(* IEC 61131-3 sources: Std_PalletMover/Class/MQTTClient_Interface (part 4) *)

            Logging_InterfLog(usLevel     :=  MQTTCLIENTINTERFACE_LOGGING_LEVEL_ERR,
                              dMsgGroup   :=  MQCLIINF_LOG_ERROR_DATAMAP_UNSUBSCRIBE_FAIL_MQCLI_GRP,
                              dMsgNbr     :=  MQCLIINF_LOG_ERROR_DATAMAP_UNSUBSCRIBE_FAIL_MQCLI_MSG,
                              pMsg        :=  MQCLIINF_LOG_ERROR_DATAMAP_UNSUBSCRIBE_FAIL_MQCLI_TEXT,
                              pPara1      :=  #tmpPara1,
                              pPara2      :=  #tmpPara2,
                              pPara3      :=  #pEntry^.pData$DINT,
                              pPara4      :=  NIL);

            pEntry^.State := DMSS_Error;
            pEntry^.udLastAction := ops.tAbsolute;

          end_if;

        //----------------------------------------------------
        //Wait for Unsubscribe confirmation
        //----------------------------------------------------
        t_e_DataMap_SubscribeStates::DMSS_WaitForUnsubscribe:

          if ops.tAbsolute - pEntry^.udLastAction >= cDataMapSubTimeout then

            //Create Log: DataMap Failed to subscribe Entry, Timeout. Moving On.

            tmpPara1 := to_dint(pEntry^.iMid);
            tmpPara2 := pEntry^.pData$DINT;

            Logging_InterfLog(usLevel     :=  MQTTCLIENTINTERFACE_LOGGING_LEVEL_ERR,
                              dMsgGroup   :=  MQCLIINF_LOG_ERROR_DATAMAP_UNSUBSCRIBE_FAIL_TIMEOUT_GRP,
                              dMsgNbr     :=  MQCLIINF_LOG_ERROR_DATAMAP_UNSUBSCRIBE_FAIL_TIMEOUT_MSG,
                              pMsg        :=  MQCLIINF_LOG_ERROR_DATAMAP_UNSUBSCRIBE_FAIL_TIMEOUT_TEXT,
                              pPara1      :=  #tmpPara1,
                              pPara2      :=  #cDataMapSubTimeout$DINT,
                              pPara3      :=  #tmpPara2,
                              pPara4      :=  NIL);

            pEntry^.State := DMSS_Unsubscribed;

          end_if;

        //----------------------------------------------------
        //Cleanup & Finish
        //----------------------------------------------------
        t_e_DataMap_SubscribeStates::DMSS_Unsubscribed:

          //Reset Mid
          pEntry^.iMid  := -1;

          //If the element must be removed do so, else return it to the original state
          if pEntry^.bRemove then

            if DataMap_RemoveElement_ByIndex( udIndex     :=  udCount,
                                              ElementType :=  DM_Subscribe) = FALSE then

               //Create Log: Failed to remove unsubscribed PubSub Entry from PubSub list.

               tmpPara1 := to_dint(pEntry^.iMid);
               tmpPara2 := to_dint(udCount);

               Logging_InterfLog(usLevel     :=  MQTTCLIENTINTERFACE_LOGGING_LEVEL_ERR,
                                 dMsgGroup   :=  MQCLIINF_LOG_ERROR_DATAMAP_UNSUBSCRIBE_FAIL_RMVE_LIST_GRP,
                                 dMsgNbr     :=  MQCLIINF_LOG_ERROR_DATAMAP_UNSUBSCRIBE_FAIL_RMVE_LIST_MSG,
                                 pMsg        :=  MQCLIINF_LOG_ERROR_DATAMAP_UNSUBSCRIBE_FAIL_RMVE_LIST_TEXT,
                                 pPara1      :=  #tmpPara1,
                                 pPara2      :=  #tmpPara2,
                                 pPara3      :=  NIL,
                                 pPara4      :=  NIL);

               pEntry^.State := DMSS_Error;
               pEntry^.udLastAction := ops.tAbsolute;

            end_if;

          //Return State to allow a resubscription.
          else

            pEntry^.State := DMSS_Ready;

          end_if;

        //----------------------------------------------------
        //Error Occurred
        //----------------------------------------------------
        t_e_DataMap_SubscribeStates::DMSS_Error:

          //Reset Mid
          pEntry^.iMid  := -1;

          //If the reset time is set, wait for reset
          if (cDataMapResetTimeout <> 0) &
             (ops.tAbsolute - pEntry^.udLastAction >= cDataMapResetTimeout) then

            pEntry^.State := DMSS_Ready;

          end_if;

      end_case;

    end_for;

  end_if;

END_FUNCTION

FUNCTION MQTTClient_Interface::DataMap_RemoveElement
	VAR_INPUT
		pElement 	: ^CHAR;
		ElementType 	: t_e_DataMap_ElementTypes;
	END_VAR
	VAR_OUTPUT
		bOK 	: BOOL;
	END_VAR
  VAR
  	udElementIndex : UDINT;
    pPublishEntry : ^t_s_DataMap_ElementEntry_Publish;
    pSubscribeEntry : ^t_s_DataMap_ElementEntry_Subscribe;
  END_VAR

  bOK := FALSE;
  udElementIndex := 0;

  if pElement = NIL then
    return;
  end_if;

  //==========================================
  //Based on the type of element
  //==========================================

  case ElementType of

    //-------------------------------------
    //Publish List
    //-------------------------------------
  	t_e_DataMap_ElementTypes::DM_Publish:

      if Config.pDataMapConfig^.udPublishElements > 0 then

        pPublishEntry := Config.pDataMapConfig^.Elements.pPublishEntries;

        for udElementIndex := 0 to Config.pDataMapConfig^.udPublishElements - 1 do

          if SigCLib.StrCmp(ps1:=#pPublishEntry^.aElement[0], ps2:=pElement) = 0 then
            bOK := DataMap_RemoveElement_ByIndex(udIndex:=udElementIndex, ElementType:=ElementType);
            exit;
          end_if;

          pPublishEntry$UDINT += sizeof(t_s_DataMap_ElementEntry_Publish);
        end_for;

      else
        return;
      end_if;

    //-------------------------------------
    //Subscribe List
    //-------------------------------------
  	t_e_DataMap_ElementTypes::DM_Subscribe:

      if Config.pDataMapConfig^.udSubscribeElements > 0 then

        pSubscribeEntry := Config.pDataMapConfig^.Elements.pSubscribeEntries;

        for udElementIndex := 0 to Config.pDataMapConfig^.udSubscribeElements - 1 do

          if SigCLib.StrCmp(ps1:=#pSubscribeEntry^.aElement[0], ps2:=pElement) = 0 then

            if pSubscribeEntry^.State = DMSS_Subscribed then
              pSubscribeEntry^.State    := DMSS_Unsubscribe;
              pSubscribeEntry^.bRemove  := TRUE;
              bOK                       := TRUE;
            end_if;

            exit;
          end_if;

          pSubscribeEntry$UDINT += sizeof(t_s_DataMap_ElementEntry_Subscribe);

        end_for;

      else
        return;
      end_if;

  end_case;

END_FUNCTION

FUNCTION MQTTClient_Interface::DataMap_RemoveElement_ByIndex
	VAR_INPUT
		udIndex 	: UDINT;
		ElementType 	: t_e_DataMap_ElementTypes;
	END_VAR
	VAR_OUTPUT
		bOK 	: BOOL;
	END_VAR
  VAR
  	tmpPara : DINT;
  END_VAR

  //Assume not OK
  bOK := FALSE;

  if Config.pDataMapConfig = NIL then
    //Create Log: Tried removing an entry from the DataMap, DataMap not inited.

    tmpPara := to_dint(udIndex);

    Logging_InterfLog(usLevel     :=  MQTTCLIENTINTERFACE_LOGGING_LEVEL_WARNING,
                      dMsgGroup   :=  MQCLIINF_LOG_WARNING_DATAMAP_REMOVE_FAILED_NOTINIT_GRP,
                      dMsgNbr     :=  MQCLIINF_LOG_WARNING_DATAMAP_REMOVE_FAILED_NOTINIT_MSG,
                      pMsg        :=  MQCLIINF_LOG_WARNING_DATAMAP_REMOVE_FAILED_NOTINIT_TEXT,
                      pPara1      :=  #tmpPara,
                      pPara2      :=  NIL,
                      pPara3      :=  NIL,
                      pPara4      :=  NIL);
    return;

  end_if;

  //========================================================
  //Based on the type of element - Find and remove the entry
  //========================================================
  case ElementType of

    //-------------------------------------
    //Publish List
    //-------------------------------------
  	t_e_DataMap_ElementTypes::DM_Publish:

      //If the index is ok
      if udIndex >= 0                                         &
         udIndex <  Config.pDataMapConfig^.udPublishElements  then

        //If this is the last entry, we don't need to copy any data
        if udIndex = Config.pDataMapConfig^.udPublishElements - 1 then

          Config.pDataMapConfig^.udPublishElements -= 1;

        //If this is not the last entry, the data has to be moved back
        else

          SigCLib.MemCpy( dst0  :=  (Config.pDataMapConfig^.Elements.pPublishEntries$UDINT + sizeof(t_s_DataMap_ElementEntry_Publish)*udIndex)$^void,
                          src0  :=  (Config.pDataMapConfig^.Elements.pPublishEntries$UDINT + sizeof(t_s_DataMap_ElementEntry_Publish)*(udIndex+1))$^void,
                          len0  :=  ((Config.pDataMapConfig^.udPublishElements-1) - udIndex)*sizeof(t_s_DataMap_ElementEntry_Publish));

          Config.pDataMapConfig^.udPublishElements -= 1;

        end_if;

        bOK := TRUE;
        return;

      else

        //Create Log: Tried removing an Entry from the DataMap with invalid Index.

        tmpPara := to_dint(udIndex);

        Logging_InterfLog(usLevel     :=  MQTTCLIENTINTERFACE_LOGGING_LEVEL_ERR,
                          dMsgGroup   :=  MQCLIINF_LOG_ERROR_DATAMAP_REMOVE_FAILED_INDEX_INV_GRP,
                          dMsgNbr     :=  MQCLIINF_LOG_ERROR_DATAMAP_REMOVE_FAILED_INDEX_INV_MSG,
                          pMsg        :=  MQCLIINF_LOG_ERROR_DATAMAP_REMOVE_FAILED_INDEX_INV_TEXT,
                          pPara1      :=  #tmpPara,
                          pPara2      :=  NIL,
                          pPara3      :=  NIL,
                          pPara4      :=  NIL);

      end_if;

    //-------------------------------------
    //Subscribe List
    //-------------------------------------
  	t_e_DataMap_ElementTypes::DM_Subscribe:

      //If the index is ok
      if udIndex >= 0 &
         udIndex <  Config.pDataMapConfig^.udSubscribeElements then

        if udIndex = Config.pDataMapConfig^.udSubscribeElements - 1 then
          Config.pDataMapConfig^.udSubscribeElements -= 1;
        else

          SigCLib.MemCpy( dst0  :=  (Config.pDataMapConfig^.Elements.pSubscribeEntries$UDINT + sizeof(t_s_DataMap_ElementEntry_Subscribe)*udIndex)$^void,
                          src0  :=  (Config.pDataMapConfig^.Elements.pSubscribeEntries$UDINT + sizeof(t_s_DataMap_ElementEntry_Subscribe)*(udIndex+1))$^void,
                          len0  :=  ((Config.pDataMapConfig^.udSubscribeElements-1) - udIndex)*sizeof(t_s_DataMap_ElementEntry_Subscribe));

          Config.pDataMapConfig^.udSubscribeElements -= 1;

        end_if;

        bOK := TRUE;
        return;

      else

        //Create Log: Tried removing an Entry from the DataMap with invalid Index.

        tmpPara := to_dint(udIndex);

        Logging_InterfLog(usLevel     :=  MQTTCLIENTINTERFACE_LOGGING_LEVEL_ERR,
                          dMsgGroup   :=  MQCLIINF_LOG_ERROR_DATAMAP_REMOVE_FAILED_INDEX_INV_GRP,
                          dMsgNbr     :=  MQCLIINF_LOG_ERROR_DATAMAP_REMOVE_FAILED_INDEX_INV_MSG,
                          pMsg        :=  MQCLIINF_LOG_ERROR_DATAMAP_REMOVE_FAILED_INDEX_INV_TEXT,
                          pPara1      :=  #tmpPara,
                          pPara2      :=  NIL,
                          pPara3      :=  NIL,
                          pPara4      :=  NIL);

      end_if;

  end_case;

END_FUNCTION

FUNCTION MQTTClient_Interface::DataMap_ResetStates
	VAR_OUTPUT
		bOK 	: BOOL;
	END_VAR
  VAR
  	udCount : UDINT;
    pSubElement : ^t_s_DataMap_ElementEntry_Subscribe;
    pPubElement : ^t_s_DataMap_ElementEntry_Publish;
  END_VAR

  //Assume Fail
  bOK := FALSE;

  //Reset Registered DataMap States
  if Config.pDataMapConfig then

    if Config.pDataMapConfig^.udSubscribeElements > 0 then
      pSubElement := Config.pDataMapConfig^.Elements.pSubscribeEntries;
      for udCount := 0 to Config.pDataMapConfig^.udSubscribeElements - 1 do
        pSubElement^.State := 0;
        pSubElement$UDINT += sizeof(t_s_DataMap_ElementEntry_Subscribe);
      end_for;
    end_if;

    if Config.pDataMapConfig^.udPublishElements > 0 then
      pPubElement:= Config.pDataMapConfig^.Elements.pPublishEntries;
      for udCount := 0 to Config.pDataMapConfig^.udPublishElements - 1 do
        pPubElement^.State := 0;
        pPubElement$UDINT += sizeof(t_s_DataMap_ElementEntry_Publish);
      end_for;
    end_if;

    bOK := TRUE;

  end_if;

END_FUNCTION

FUNCTION MQTTClient_Interface::DataMap_Return_Callback
	VAR_INPUT
		pThis 	: ^void;
		MsgType 	: MQTTClient_Interface::t_e_PubSubRetCodes;
		iMid 	: INT;
		iGrantedQoS 	: INT;
		pMessage 	: ^MQTTClient::t_s_MQTTMessage;
	END_VAR

  //Call Internal Method
  pThis$^MQTTClient_Interface^.DataMap_Return(MsgType     :=  MsgType,
                                              iMid        :=  iMid,
                                              iGrantedQoS :=  iGrantedQoS,
                                              pMessage    :=  pMessage);

END_FUNCTION

FUNCTION MQTTClient_Interface::DataMap_Clear

  if Config.pDataMapConfig                             &
     Config.pDataMapConfig^.Elements.pPublishEntries   &
     Config.pDataMapConfig^.Elements.pSubscribeEntries then

    Config.pDataMapConfig^.udPublishElements := 0;
    Config.pDataMapConfig^.udSubscribeElements := 0;

    sigclib_memset( dst :=  Config.pDataMapConfig^.Elements.pPublishEntries,
                    c   :=  0x00,
                    len :=  sizeof(t_s_DataMap_ElementEntry_Publish)*Config.pDataMapConfig^.udEntries);

    sigclib_memset( dst :=  Config.pDataMapConfig^.Elements.pSubscribeEntries,
                    c   :=  0x00,
                    len :=  sizeof(t_s_DataMap_ElementEntry_Subscribe)*Config.pDataMapConfig^.udEntries);

  end_if;

END_FUNCTION

FUNCTION MQTTClient_Interface::DataMap_Return
	VAR_INPUT
		MsgType 	: MQTTClient_Interface::t_e_PubSubRetCodes;
		iMid 	: INT;
		iGrantedQoS 	: INT;
		pMessage 	: ^MQTTClient::t_s_MQTTMessage;
	END_VAR
  VAR
  	udCount         : UDINT;
  	pArray          : ^void;
    pArrEntry       : ^void;
    udNumSubEntries : UDINT;
    pSubEntry       : ^t_s_DataMap_ElementEntry_Subscribe;
    pPubEntry       : ^t_s_DataMap_ElementEntry_Publish;
    bFound          : BOOL;
    udCopyLen       : UDINT;
    tmpPara1        : DINT;
    tmpPara2        : DINT;
    tmpPara3        : DINT;
    tmpPara4        : DINT;
    tmpData         : DINT; //Variable to contain the received 4 byte values temporarily, this avoids writing rubbish on the server
  END_VAR

  //Clear pSubEntries Pointer, Memory is malloc'd and set to this pointer if MsgType = PSRC_PublishReceived,
  //All exit paths must be observed to avoid a memory leak here.
  pArray := NIL;

  if Config.pDataMapConfig = NIL then
    //Create Log: Received Datamap Callback for DataMap Whilst DataMap is not Inited.

    tmpPara1 := to_dint(iMid);

    if pMessage <> NIL then
      tmpPara2 := to_dint(pMessage^.mid);
    else
      tmpPara2 := 16#FFFF;
    end_if;

    Logging_InterfLog(usLevel     :=  MQTTCLIENTINTERFACE_LOGGING_LEVEL_WARNING,
                      dMsgGroup   :=  MQCLIINF_LOG_WARNING_DATAMAP_CALLBACK_MAP_NOTINIT_GRP,
                      dMsgNbr     :=  MQCLIINF_LOG_WARNING_DATAMAP_CALLBACK_MAP_NOTINIT_MSG,
                      pMsg        :=  MQCLIINF_LOG_WARNING_DATAMAP_CALLBACK_MAP_NOTINIT_TEXT,
                      pPara1      :=  #tmpPara1,
                      pPara2      :=  #tmpPara2,
                      pPara3      :=  NIL,
                      pPara4      :=  NIL);

    return;
  end_if;

  bFound := FALSE;

  //======================================
  //Find the DataMap Entry with this Mid
  //======================================
  case MsgType of

    //------------------------------------------------
    //Disconnected
    //------------------------------------------------
  	PSRC_Disconnected:

      //Reset all the DataMap Entries

      return;

    //---------------------------------------------------------------------------
    //Subscribe Related, can only be: one entry (Mid Tracked) or all (Mid = -1)
    //---------------------------------------------------------------------------
  	PSRC_Subscribed, PSRC_Unsubscribed:

      pSubEntry := Config.pDataMapConfig^.Elements.pSubscribeEntries;
      if Config.pDataMapConfig^.udSubscribeElements > 0 then

        //If this is an unsubscribe all (iMid=-1), then simply unsubscribe all and return,
        //else find the entry to unsubscribe
        if iMid = -1 then

          for udCount := 0 to Config.pDataMapConfig^.udSubscribeElements - 1 do
            pSubEntry^.State := DMSS_Unsubscribed;
            pSubEntry$UDINT += sizeof(t_s_DataMap_ElementEntry_Subscribe);
          end_for;
          return;

        //This is a specific entry, step over all entries to find the matching entry.
        else

          for udCount := 0 to Config.pDataMapConfig^.udSubscribeElements - 1 do
            if pSubEntry^.iMid = iMid then
              bFound := TRUE;
              exit;
            end_if;
            pSubEntry$UDINT += sizeof(t_s_DataMap_ElementEntry_Subscribe);
          end_for;

        end_if;
      end_if;

    //----------------------------------------------------
    //Publish Related, Mid tracked, can only be one entry
    //----------------------------------------------------
  	PSRC_Published:

      pPubEntry := Config.pDataMapConfig^.Elements.pPublishEntries;
      for udCount := 0 to Config.pDataMapConfig^.udEntries - 1 do
        if pPubEntry^.iMid = iMid then
          pPubEntry^.iMid := -1;
          bFound := TRUE;
          exit;
        end_if;
        pPubEntry$UDINT += sizeof(t_s_DataMap_ElementEntry_Publish);
      end_for;

    //-------------------------------------------------------------------
    //Subscribe Related, Use Topic for relation, can be multiple entries
    //-------------------------------------------------------------------
    PSRC_PublishReceived:

      pArray := MQTTClient.MallocV1(size0 :=  sizeof(^void) * Config.pPubSubConfig^.PubSubList.udMaxEntries,
                                    mark0 :=  MQTTCLIENTINTERFACE_DEFAULT_MALLOC_MARK);

      //If the Malloc succeeded
      if pArray <> NIL then

        SigCLib.MemSet( dst :=  pArray,
                        c   :=  0x00,
                        len :=  sizeof(^void) * Config.pPubSubConfig^.PubSubList.udMaxEntries);

        udNumSubEntries := 0;
        pSubEntry := Config.pDataMapConfig^.Elements.pSubscribeEntries;
        pArrEntry := pArray;

        for udCount := 0 to Config.pDataMapConfig^.udSubscribeElements - 1 do

          //If this is not a stale entry and the topic matches, add to the list.
          if PubSub_TopicCompare(pStr:=pMessage^.topic, pWCString:=#pSubEntry^.aTopic[0]) then

            bFound := TRUE;
            pArrEntry^$UDINT := pSubEntry$UDINT;
            pArrEntry$UDINT += sizeof(^void);
            udNumSubEntries += 1;

          end_if;

          pSubEntry$UDINT += sizeof(t_s_DataMap_ElementEntry_Subscribe);

        end_for;

      //Malloc failed, we won't be able to deliver the message to the Application, report error.
      else

        tmpPara1 := to_dint(iMid);

        if pMessage <> NIL then
          tmpPara2 := to_dint(pMessage^.mid);
        else
          tmpPara2 := 16#FFFF;
        end_if;

        Logging_InterfLog(usLevel     :=  MQTTCLIENTINTERFACE_LOGGING_LEVEL_ERR,
                          dMsgGroup   :=  MQCLIINF_LOG_ERROR_DATAMAP_RETURN_NOMEM_ARRAY_GRP,
                          dMsgNbr     :=  MQCLIINF_LOG_ERROR_DATAMAP_RETURN_NOMEM_ARRAY_MSG,
                          pMsg        :=  MQCLIINF_LOG_ERROR_DATAMAP_RETURN_NOMEM_ARRAY_TEXT,
                          pPara1      :=  #tmpPara1,
                          pPara2      :=  #tmpPara2,
                          pPara3      :=  NIL,
                          pPara4      :=  NIL);

        return;

      end_if;

  end_case;

  if bFound = FALSE then
    //Create Log: Received DataMap Callback but did not find corresponding entry.

    tmpPara1 := to_dint(iMid);

    if pMessage <> NIL then
      tmpPara2 := to_dint(pMessage^.mid);
    else
      tmpPara2 := 16#FFFF;
    end_if;

    Logging_InterfLog(usLevel     :=  MQTTCLIENTINTERFACE_LOGGING_LEVEL_ERR,
                      dMsgGroup   :=  MQCLIINF_LOG_WARNING_DATAMAP_CALLBACK_ENTRY_NOTFOUND_GRP,
                      dMsgNbr     :=  MQCLIINF_LOG_WARNING_DATAMAP_CALLBACK_ENTRY_NOTFOUND_MSG,
                      pMsg        :=  MQCLIINF_LOG_WARNING_DATAMAP_CALLBACK_ENTRY_NOTFOUND_TEXT,
                      pPara1      :=  #tmpPara1,
                      pPara2      :=  #tmpPara2,
                      pPara3      :=  NIL,
                      pPara4      :=  NIL);

    //If the pSubEntries Pointer is set, free
    if pArray then
      MQTTClient.Free(mptr:=pArray);
      pArray := NIL;
    end_if;

    return;
  end_if;

  //=====================================================
  //Based on the type of message, edit the DataMap
  //=====================================================
  case MsgType of

    //------------------------------------------------
    //Subscribe completed, check and advance
    //------------------------------------------------
    t_e_PubSubRetCodes::PSRC_Subscribed:

      //if the QoS is invalid, set state and log
      if iGrantedQoS < MQTT_PROT_QOS_MIN |
         iGrantedQoS > MQTT_PROT_QOS_MAX then
        //Create Log: DataMap Element Failed to Subscribe, Returned QoS Invalid, Element=XXXX Granted=XX, Requested=XX

        tmpPara1 := to_dint(iMid);

        if pMessage <> NIL then
          tmpPara2 := to_dint(pMessage^.mid);
        else
          tmpPara2 := 16#FFFF;
        end_if;

        tmpPara3 := to_dint(iGrantedQoS);

        if pSubEntry <> NIL then
          tmpPara4 := to_dint(pSubEntry^.iQoS);
        else
          tmpPara4 := 16#FFFF;
        end_if;

        Logging_InterfLog(usLevel     :=  MQTTCLIENTINTERFACE_LOGGING_LEVEL_ERR,
                          dMsgGroup   :=  MQCLIINF_LOG_ERROR_DATAMAP_SUB_CONF_WRONG_QOS_GRP,
                          dMsgNbr     :=  MQCLIINF_LOG_ERROR_DATAMAP_SUB_CONF_WRONG_QOS_MSG,
                          pMsg        :=  MQCLIINF_LOG_ERROR_DATAMAP_SUB_CONF_WRONG_QOS_TEXT,
                          pPara1      :=  #tmpPara1,
                          pPara2      :=  #tmpPara2,
                          pPara3      :=  #tmpPara3,
                          pPara4      :=  #tmpPara4);

        pSubEntry^.State := DMSS_Error;
        return;
      end_if;

      //If the Entry is not in the correct state
      if pSubEntry^.State <> DMSS_WaitForSubscribe then
        //Create Log: DataMap Element failed to Subscribe, Subscription returned valid but the Element State was invalid, Element=XXXX, Granted QoS=XX

        tmpPara1 := to_dint(iMid);

        if pMessage <> NIL then
          tmpPara2 := to_dint(pMessage^.mid);
        else
          tmpPara2 := 16#FFFF;
        end_if;

        tmpPara3 := to_dint(pSubEntry^.State);

        Logging_InterfLog(usLevel     :=  MQTTCLIENTINTERFACE_LOGGING_LEVEL_ERR,
                          dMsgGroup   :=  MQCLIINF_LOG_WARNING_DATAMAP_SUB_CONFD_WRONG_STATE_GRP,
                          dMsgNbr     :=  MQCLIINF_LOG_WARNING_DATAMAP_SUB_CONFD_WRONG_STATE_MSG,
                          pMsg        :=  MQCLIINF_LOG_WARNING_DATAMAP_SUB_CONFD_WRONG_STATE_TEXT,
                          pPara1      :=  #tmpPara1,
                          pPara2      :=  #tmpPara2,
                          pPara3      :=  #tmpPara3,
                          pPara4      :=  NIL);

        pSubEntry^.State := DMSS_Error;
        return;

      end_if;

      //If QoS does not match then log the difference and update
      if iGrantedQoS <> pSubEntry^.iQoS then
        //Create Log: DataMap Element Granted QoS differs from Requested, Element=XXXX Granted=XX, Requested=XX

        tmpPara1 := to_dint(iMid);

        if pMessage <> NIL then
          tmpPara2 := to_dint(pMessage^.mid);
        else
          tmpPara2 := 16#FFFF;
        end_if;

        tmpPara3 := to_dint(iGrantedQoS);

        if pSubEntry <> NIL then
          tmpPara4 := to_dint(pSubEntry^.iQoS);
        else
          tmpPara4 := 16#FFFF;
        end_if;

        Logging_InterfLog(usLevel     :=  MQTTCLIENTINTERFACE_LOGGING_LEVEL_INFO,
                          dMsgGroup   :=  MQCLIINF_LOG_INFO_DATAMAP_SUB_CONFD_QOS_DIFFERS_GRP,
                          dMsgNbr     :=  MQCLIINF_LOG_INFO_DATAMAP_SUB_CONFD_QOS_DIFFERS_MSG,
                          pMsg        :=  MQCLIINF_LOG_INFO_DATAMAP_SUB_CONFD_QOS_DIFFERS_TEXT,
                          pPara1      :=  #tmpPara1,
                          pPara2      :=  #tmpPara2,
                          pPara3      :=  #tmpPara3,
                          pPara4      :=  #tmpPara4);

        pSubEntry^.iQoS := iGrantedQoS;
      end_if;

      pSubEntry^.State := DMSS_Subscribed;

    //------------------------------------------------
    //Unsubscribe completed, check and advance
    //------------------------------------------------
    t_e_PubSubRetCodes::PSRC_Unsubscribed:

      //Create Log: DataMap Element Unsubscribed, Element=XXXX

      tmpPara1 := to_dint(iMid);

      if pMessage <> NIL then
        tmpPara2 := to_dint(pMessage^.mid);
      else
        tmpPara2 := 16#FFFF;
      end_if;

      Logging_InterfLog(usLevel     :=  MQTTCLIENTINTERFACE_LOGGING_LEVEL_INFO,
                        dMsgGroup   :=  MQCLIINF_LOG_INFO_DATAMAP_UNSUB_CONFD_GRP,
                        dMsgNbr     :=  MQCLIINF_LOG_INFO_DATAMAP_UNSUB_CONFD_MSG,
                        pMsg        :=  MQCLIINF_LOG_INFO_DATAMAP_UNSUB_CONFD_TEXT,
                        pPara1      :=  #tmpPara1,
                        pPara2      :=  #tmpPara2,
                        pPara3      :=  NIL,
                        pPara4      :=  NIL);

      pSubEntry^.State := DMSS_Unsubscribed;

    //------------------------------------------------
    //Publish Received, Set Data
    //------------------------------------------------
    t_e_PubSubRetCodes::PSRC_PublishReceived:

      if pMessage then

        //Step over all the entries found and process the message
        if udNumSubEntries > 0 then

          for udCount := 0 to udNumSubEntries - 1 do

            //pSubEntry := aSubEntries[udCount];
            pSubEntry$UDINT := (pArray$UDINT + sizeof(^void)*udCount);
            pSubEntry := pSubEntry^$^t_s_DataMap_ElementEntry_Subscribe;

            //======================================
            //Set the data based on the type
            //======================================
            case pSubEntry^.DataType of
              //----------------------
              //4 Bytes
              //----------------------
              t_e_DataMap_DataTypes::DD_UDINT:

                udCopyLen := pMessage^.payloadlen;

                if udCopyLen > sizeof(UDINT) then
                  //Create Log: More data received than is able to be fit into Datamap element, data truncated

                  tmpPara1 := to_dint(iMid);

                  if pMessage <> NIL then
                    tmpPara2 := to_dint(pMessage^.mid);
                  else
                    tmpPara2 := 16#FFFF;
                  end_if;

                  Logging_InterfLog(usLevel     :=  MQTTCLIENTINTERFACE_LOGGING_LEVEL_WARNING,
                                    dMsgGroup   :=  MQCLIINF_LOG_WARNING_DATAMAP_DATA_TRUNCATED_UDINT_GRP,
                                    dMsgNbr     :=  MQCLIINF_LOG_WARNING_DATAMAP_DATA_TRUNCATED_UDINT_MSG,
                                    pMsg        :=  MQCLIINF_LOG_WARNING_DATAMAP_DATA_TRUNCATED_UDINT_TEXT,
                                    pPara1      :=  #tmpPara1,
                                    pPara2      :=  #tmpPara2,
                                    pPara3      :=  #udCopyLen$DINT,
                                    pPara4      :=  NIL);

                  udCopyLen := sizeof(UDINT);

                end_if;

                tmpData := 0;
                SigCLib.MemCpy( dst0  :=  #tmpData,
                                src0  :=  pMessage^.payload,
                                len0  :=  pMessage^.payloadlen);

                WR( pt    :=  pSubEntry^.pData,
                    dData :=  tmpData$DINT);

              //----------------------
              //4 Bytes
              //----------------------
              t_e_DataMap_DataTypes::DD_DINT:

                udCopyLen := pMessage^.payloadlen;

                if udCopyLen > sizeof(DINT) then
                  //Create Log: More data received than is able to be fit into Datamap element, data truncated

                  tmpPara1 := to_dint(iMid);

                  if pMessage <> NIL then
                    tmpPara2 := to_dint(pMessage^.mid);
                  else
                    tmpPara2 := 16#FFFF;
                  end_if;

                  Logging_InterfLog(usLevel     :=  MQTTCLIENTINTERFACE_LOGGING_LEVEL_WARNING,
                                    dMsgGroup   :=  MQCLIINF_LOG_WARNING_DATAMAP_DATA_TRUNCATED_DINT_GRP,
                                    dMsgNbr     :=  MQCLIINF_LOG_WARNING_DATAMAP_DATA_TRUNCATED_DINT_MSG,
                                    pMsg        :=  MQCLIINF_LOG_WARNING_DATAMAP_DATA_TRUNCATED_DINT_TEXT,
                                    pPara1      :=  #tmpPara1,
                                    pPara2      :=  #tmpPara2,
                                    pPara3      :=  #udCopyLen$DINT,
                                    pPara4      :=  NIL);

                  udCopyLen := sizeof(UDINT);

                end_if;

                tmpData := 0;
                SigCLib.MemCpy( dst0  :=  #tmpData,
                                src0  :=  pMessage^.payload,
                                len0  :=  pMessage^.payloadlen);

                WR( pt    :=  pSubEntry^.pData,
                    dData :=  tmpData$DINT);

              //----------------------
              //4 Bytes
              //----------------------
              t_e_DataMap_DataTypes::DD_REAL:

                udCopyLen := pMessage^.payloadlen;

                if udCopyLen > sizeof(REAL) then
                  //Create Log: More data received than is able to be fit into Datamap element, data truncated

                  tmpPara1 := to_dint(iMid);

                  if pMessage <> NIL then
                    tmpPara2 := to_dint(pMessage^.mid);
                  else
                    tmpPara2 := 16#FFFF;
                  end_if;

                  Logging_InterfLog(usLevel     :=  MQTTCLIENTINTERFACE_LOGGING_LEVEL_WARNING,
                                    dMsgGroup   :=  MQCLIINF_LOG_WARNING_DATAMAP_DATA_TRUNCATED_REAL_GRP,
                                    dMsgNbr     :=  MQCLIINF_LOG_WARNING_DATAMAP_DATA_TRUNCATED_REAL_MSG,
                                    pMsg        :=  MQCLIINF_LOG_WARNING_DATAMAP_DATA_TRUNCATED_REAL_TEXT,
                                    pPara1      :=  #tmpPara1,
                                    pPara2      :=  #tmpPara2,
                                    pPara3      :=  #udCopyLen$DINT,
                                    pPara4      :=  NIL);

                  udCopyLen := sizeof(UDINT);

                end_if;

                tmpData := 0;
                SigCLib.MemCpy( dst0  :=  #tmpData,
                                src0  :=  pMessage^.payload,
                                len0  :=  pMessage^.payloadlen);

                WR( pt    :=  pSubEntry^.pData,
                    dData :=  tmpData$DINT);

              //----------------------
              //Dynamic Size
              //----------------------
              t_e_DataMap_DataTypes::DD_String:

                pSubEntry^.pData$^StringInternal^.WriteDataOff(udLen :=  pMessage^.payloadlen,
                                                               udOff :=  0,
                                                               pData :=  pMessage^.payload$^USINT);

            end_case;

          end_for;

        end_if;

      else

        //Create Log: DataMap Received PublishReceived Callback from MQTTClientInterface but no message was set

        tmpPara1 := to_dint(iMid);

        if pMessage <> NIL then
          tmpPara2 := to_dint(pMessage^.mid);
        else
          tmpPara2 := 16#FFFF;
        end_if;

        Logging_InterfLog(usLevel     :=  MQTTCLIENTINTERFACE_LOGGING_LEVEL_WARNING,
                          dMsgGroup   :=  MQCLIINF_LOG_WARNING_DATAMAP_DATA_EMPTY_GRP,
                          dMsgNbr     :=  MQCLIINF_LOG_WARNING_DATAMAP_DATA_EMPTY_MSG,
                          pMsg        :=  MQCLIINF_LOG_WARNING_DATAMAP_DATA_EMPTY_TEXT,
                          pPara1      :=  #tmpPara1,
                          pPara2      :=  #tmpPara2,
                          pPara3      :=  NIL,
                          pPara4      :=  NIL);

      end_if;

      //If the pSubEntries Pointer is set, free
      if pArray then
        MQTTClient.Free(mptr:=pArray);
        pArray := NIL;
      end_if;

    //------------------------------------------------
    //Publish Complete
    //------------------------------------------------
    t_e_PubSubRetCodes::PSRC_Published:

      pPubEntry^.bPublishComplete := TRUE;

      return;

  end_case;

END_FUNCTION

//================================================================================================================================================================
//-------------------------------------------------------------------END OF DATAMAP METHODS-----------------------------------------------------------------------
//================================================================================================================================================================

//================================================================================================================================================================
//------------------------------------------------------------------------CALLBACK METHODS------------------------------------------------------------------------
//================================================================================================================================================================
FUNCTION MQTTClient_Interface::Callback_OnConnectWithFlags
	VAR_INPUT
		pThis 	: ^void;
		retCode 	: INT;
    flags   : BYTE;
	END_VAR

  if pThis then
    pThis$^MQTTClient_Interface^.OnConnectWithFlags(retCode:=retCode,flags:=flags);
  end_if;

END_FUNCTION

FUNCTION MQTTClient_Interface::Callback_OnDisconnect
	VAR_INPUT
		pThis 	: ^void;
		retCode 	: INT;
	END_VAR

  if pThis then
    pThis$^MQTTClient_Interface^.OnDisconnect(retCode:=retCode);
  end_if;

END_FUNCTION

FUNCTION MQTTClient_Interface::Callback_OnPublish
	VAR_INPUT
		pThis 	: ^void;
		mid 	: INT;
	END_VAR

  if pThis then
    pThis$^MQTTClient_Interface^.OnPublish(mid:=mid);
  end_if;

END_FUNCTION

FUNCTION MQTTClient_Interface::Callback_OnMessage
	VAR_INPUT
		pThis 	: ^void;
		pMessage 	: ^MQTTClient::t_s_MQTTMessage;
	END_VAR

  if pThis then
    pThis$^MQTTClient_Interface^.OnMessage(pMessage:=pMessage);
  end_if;

END_FUNCTION

FUNCTION MQTTClient_Interface::Callback_OnSubscribe
	VAR_INPUT
		pThis 	: ^void;
		mid 	: INT;
		qos_count 	: INT;
		granted_qos 	: ^INT;
	END_VAR

  if pThis then
    pThis$^MQTTClient_Interface^.OnSubscribe( mid         :=  mid,
                                              qos_count   := qos_count,
                                              granted_qos := granted_qos);
  end_if;

END_FUNCTION

FUNCTION MQTTClient_Interface::Callback_OnUnsubscribe
	VAR_INPUT
		pThis 	: ^void;
		mid 	: INT;
	END_VAR

  if pThis then
    pThis$^MQTTClient_Interface^.OnUnsubscribe(mid:=mid);
  end_if;

END_FUNCTION

FUNCTION MQTTClient_Interface::Callback_OnLog
	VAR_INPUT
		pThis 	: ^void;
		level 	: INT;
		pStr 	: ^CHAR;
	END_VAR

  if pThis then
    pThis$^MQTTClient_Interface^.OnLog( level :=  level,
                                        pStr  :=  pStr);
  end_if;

END_FUNCTION

FUNCTION MQTTClient_Interface::Callback_OnLog_WithDetail
	VAR_INPUT
		pThis 	    : ^void;
		usLevel 	  : USINT;
		dMsgGroup 	: DINT;
		dMsgNbr 	  : DINT;
		pMsg 	      : ^CHAR;
		pPara1 	    : ^DINT;
		pPara2 	    : ^DINT;
		pPara3 	    : ^DINT;
		pPara4 	    : ^DINT;
	END_VAR

  if pThis then

    pThis$^MQTTClient_Interface^.OnLog_WithDetail(usLevel   := usLevel,
                                                  dMsgGroup := dMsgGroup,
                                                  dMsgNbr   := dMsgNbr,
                                                  pMsg      := pMsg,
                                                  pPara1    := pPara1,
                                                  pPara2    := pPara2,
                                                  pPara3    := pPara3,
                                                  pPara4    := pPara4);

  end_if;

END_FUNCTION

FUNCTION MQTTClient_Interface::OnConnectWithFlags
	VAR_INPUT
		retCode 	: INT;
		flags 	  : BYTE;
	END_VAR
  VAR
  	tmpPara, tmpPara2 : DINT;
  END_VAR

  //=================================
  //Internal Actions

  //If in the correct state, process the Connect message, else log
  if InterfaceState = MCIS_WaitForConnection |
     InterfaceState = MCIS_Reconnecting      then

    if retCode = MQTT_PROT_CONNACK_RET_CONNACCEPTED then

      InterfaceState := MCIS_Connected;

      //Handle Flags

        //Tell the Subscribed entities that they have been unsubscribed.
        if  SessionPresent.Read() = 0 then
          MQTT_SetCleanSession();
        end_if;

      //Create Log: Connected

      tmpPara := to_dint(retCode);
      tmpPara2 := to_dint(flags);

      Logging_InterfLog(usLevel     :=  MQTTCLIENTINTERFACE_LOGGING_LEVEL_INFO,
                        dMsgGroup   :=  MQCLIINF_LOG_INFO_CONNECTION_CONNECTED_GRP,
                        dMsgNbr     :=  MQCLIINF_LOG_INFO_CONNECTION_CONNECTED_MSG,
                        pMsg        :=  MQCLIINF_LOG_INFO_CONNECTION_CONNECTED_TEXT,
                        pPara1      :=  #tmpPara,
                        pPara2      :=  #tmpPara2,
                        pPara3      :=  NIL,
                        pPara4      :=  NIL);

      Diagnostic_Event( Event   :=  DL_Connect,
                        udValue :=  0);

    elsif retCode = MQTT_PROT_CONNACK_RET_PROTVERSION then

      //Create Log: Connection Failed, Protocol Versions Mismatch

      tmpPara := to_dint(retCode);

      Logging_InterfLog(usLevel     :=  MQTTCLIENTINTERFACE_LOGGING_LEVEL_ERR,
                        dMsgGroup   :=  MQCLIINF_LOG_ERROR_CONNECTION_CONN_FAIL_VER_GRP,
                        dMsgNbr     :=  MQCLIINF_LOG_ERROR_CONNECTION_CONN_FAIL_VER_MSG,
                        pMsg        :=  MQCLIINF_LOG_ERROR_CONNECTION_CONN_FAIL_VER_TEXT,
                        pPara1      :=  #tmpPara,
                        pPara2      :=  NIL,
                        pPara3      :=  NIL,
                        pPara4      :=  NIL);

      InterfaceState := MCIS_Error;

    elsif retCode = MQTT_PROT_CONNACK_RET_ID_REJECTED then

      //Create Log: Connection Failed, ClientID Rejected

      tmpPara := to_dint(retCode);

      Logging_InterfLog(usLevel     :=  MQTTCLIENTINTERFACE_LOGGING_LEVEL_ERR,
                        dMsgGroup   :=  MQCLIINF_LOG_ERROR_CONNECTION_CONN_FAIL_CLIENTID_GRP,
                        dMsgNbr     :=  MQCLIINF_LOG_ERROR_CONNECTION_CONN_FAIL_CLIENTID_MSG,
                        pMsg        :=  MQCLIINF_LOG_ERROR_CONNECTION_CONN_FAIL_CLIENTID_TEXT,
                        pPara1      :=  #tmpPara,
                        pPara2      :=  NIL,
                        pPara3      :=  NIL,
                        pPara4      :=  NIL);

      InterfaceState := MCIS_Error;

    elsif retCode = MQTT_PROT_CONNACK_RET_SERVER_UNAVAIL then

      //Create Log: Connection Failed, Server unavailable

      tmpPara := to_dint(retCode);

      Logging_InterfLog(usLevel     :=  MQTTCLIENTINTERFACE_LOGGING_LEVEL_ERR,
                        dMsgGroup   :=  MQCLIINF_LOG_ERROR_CONNECTION_CONN_FAIL_SERV_UNAV_GRP,
                        dMsgNbr     :=  MQCLIINF_LOG_ERROR_CONNECTION_CONN_FAIL_SERV_UNAV_MSG,
                        pMsg        :=  MQCLIINF_LOG_ERROR_CONNECTION_CONN_FAIL_SERV_UNAV_TEXT,
                        pPara1      :=  #tmpPara,
                        pPara2      :=  NIL,
                        pPara3      :=  NIL,
                        pPara4      :=  NIL);

      InterfaceState := MCIS_Error;

    elsif retCode = MQTT_PROT_CONNACK_RET_USN_PASS then

      //Create Log: Connection Failed, Username and/or Password incorrect

      tmpPara := to_dint(retCode);

      Logging_InterfLog(usLevel     :=  MQTTCLIENTINTERFACE_LOGGING_LEVEL_ERR,
                        dMsgGroup   :=  MQCLIINF_LOG_ERROR_CONNECTION_CONN_FAIL_USNPWD_GRP,
                        dMsgNbr     :=  MQCLIINF_LOG_ERROR_CONNECTION_CONN_FAIL_USNPWD_MSG,
                        pMsg        :=  MQCLIINF_LOG_ERROR_CONNECTION_CONN_FAIL_USNPWD_TEXT,
                        pPara1      :=  #tmpPara,
                        pPara2      :=  NIL,
                        pPara3      :=  NIL,
                        pPara4      :=  NIL);

      InterfaceState := MCIS_Error;

    elsif retCode = MQTT_PROT_CONNACK_RET_NOT_AUTHD then

      //Create Log: Connection Failed, Not authorised

      tmpPara := to_dint(retCode);

      Logging_InterfLog(usLevel     :=  MQTTCLIENTINTERFACE_LOGGING_LEVEL_ERR,
                        dMsgGroup   :=  MQCLIINF_LOG_ERROR_CONNECTION_CONN_FAIL_NOT_AUTH_GRP,
                        dMsgNbr     :=  MQCLIINF_LOG_ERROR_CONNECTION_CONN_FAIL_NOT_AUTH_MSG,
                        pMsg        :=  MQCLIINF_LOG_ERROR_CONNECTION_CONN_FAIL_NOT_AUTH_TEXT,
                        pPara1      :=  #tmpPara,
                        pPara2      :=  NIL,
                        pPara3      :=  NIL,
                        pPara4      :=  NIL);

      InterfaceState := MCIS_Error;

    end_if;

  //Not expecting callback
  else

    //Create Log: Unexpected Connect Callback Received

    tmpPara := to_dint(retCode);

    Logging_InterfLog(usLevel     :=  MQTTCLIENTINTERFACE_LOGGING_LEVEL_ERR,
                      dMsgGroup   :=  MQCLIINF_LOG_WARNING_CONNECTION_CONN_CALLBACK_UNEXP_GRP,
                      dMsgNbr     :=  MQCLIINF_LOG_WARNING_CONNECTION_CONN_CALLBACK_UNEXP_MSG,
                      pMsg        :=  MQCLIINF_LOG_WARNING_CONNECTION_CONN_CALLBACK_UNEXP_TEXT,
                      pPara1      :=  #tmpPara,
                      pPara2      :=  NIL,
                      pPara3      :=  NIL,
                      pPara4      :=  NIL);

  end_if;

  //=================================
  //Signed in Objects

END_FUNCTION

FUNCTION MQTTClient_Interface::OnDisconnect
	VAR_INPUT
		retCode 	: INT;
	END_VAR
  VAR
  	udCount : UDINT;
    tmpPara : DINT;
    pEntry  : ^t_s_PubSubEntry;
  END_VAR

  //=================================
  //Internal Actions

  //=============================================
  //Handle Disconnect Message according to state
  //=============================================
  case InterfaceState of

    //------------------------------------------------------------------
    //Was Connected and then Disconnected, advance State
    //------------------------------------------------------------------
  	MQTTClient_Interface::t_e_MQTTClientStates::MCIS_Connected:

      //User Request, Go to ready
      if retCode = MQTTCLIENT_DISCONNECT_RETCODE_USER then

        InterfaceState := MCIS_Ready;
        //Create Log: MQTT Interface Successfully Disconnected due to user request

        tmpPara := to_dint(retcode);

        Logging_InterfLog(usLevel     :=  MQTTCLIENTINTERFACE_LOGGING_LEVEL_INFO,
                          dMsgGroup   :=  MQCLIINF_LOG_INFO_CONNECTION_DISCONNECTED_GRP,
                          dMsgNbr     :=  MQCLIINF_LOG_INFO_CONNECTION_DISCONNECTED_MSG,
                          pMsg        :=  MQCLIINF_LOG_INFO_CONNECTION_DISCONNECTED_TEXT,
                          pPara1      :=  #tmpPara,
                          pPara2      :=  NIL,
                          pPara3      :=  NIL,
                          pPara4      :=  NIL);

      //Unexpected, wait for connection
      elsif retCode = MQTTCLIENT_DISCONNECT_RETCODE_UNEXP then

        InterfaceState := MCIS_Reconnecting;
        //Diagnostic Info:
        Diagnostic_Event( Event   :=  DL_ConnectRetry,
                          udValue :=  0);

        //Create Log: MQTT Interface Disconnected Unexpectedly, Waiting for reconnection.

        tmpPara := to_dint(retcode);

        Logging_InterfLog(usLevel     :=  MQTTCLIENTINTERFACE_LOGGING_LEVEL_WARNING,
                          dMsgGroup   :=  MQCLIINF_LOG_ERROR_CONNECTION_DISCONN_UNEXP_GRP,
                          dMsgNbr     :=  MQCLIINF_LOG_ERROR_CONNECTION_DISCONN_UNEXP_MSG,
                          pMsg        :=  MQCLIINF_LOG_ERROR_CONNECTION_DISCONN_UNEXP_TEXT,
                          pPara1      :=  #tmpPara,
                          pPara2      :=  NIL,
                          pPara3      :=  NIL,
                          pPara4      :=  NIL);

      //Undefined RetCode, Log, Error
      else

        //Create Log: MQTT Client Diconnected with undefined disconnect code.

        tmpPara := to_dint(retcode);

        Logging_InterfLog(usLevel     :=  MQTTCLIENTINTERFACE_LOGGING_LEVEL_ERR,
                          dMsgGroup   :=  MQCLIINF_LOG_ERROR_CONNECTION_DISCONN_UNKNOWN_CODE_GRP,
                          dMsgNbr     :=  MQCLIINF_LOG_ERROR_CONNECTION_DISCONN_UNKNOWN_CODE_MSG,
                          pMsg        :=  MQCLIINF_LOG_ERROR_CONNECTION_DISCONN_UNKNOWN_CODE_TEXT,
                          pPara1      :=  #tmpPara,
                          pPara2      :=  NIL,
                          pPara3      :=  NIL,
                          pPara4      :=  NIL);

        InterfaceState := MCIS_Error;

      end_if;

    //------------------------------------------------------------------
    //Unexpected callback
    //------------------------------------------------------------------
    else

      //Create Log: Unexpected Disconnect Message Received from MQTT Client

      tmpPara := to_dint(retcode);

      Logging_InterfLog(usLevel     :=  MQTTCLIENTINTERFACE_LOGGING_LEVEL_WARNING,
                        dMsgGroup   :=  MQCLIINF_LOG_WARNING_CONNECTION_DISCONN_CALLBACK_UNEXP_GRP,
                        dMsgNbr     :=  MQCLIINF_LOG_WARNING_CONNECTION_DISCONN_CALLBACK_UNEXP_MSG,
                        pMsg        :=  MQCLIINF_LOG_WARNING_CONNECTION_DISCONN_CALLBACK_UNEXP_TEXT,
                        pPara1      :=  #tmpPara,
                        pPara2      :=  NIL,
                        pPara3      :=  NIL,
                        pPara4      :=  NIL);

      InterfaceState := MCIS_Error;

  end_case;

  //Perform the disconnect callbacks for the items in the pubsub list
  if Config.pPubSubConfig &
     Config.pPubSubConfig^.PubSubList.udNumEntries > 0 then

    for udCount := 0 to Config.pPubSubConfig^.PubSubList.udNumEntries -1 do

      pEntry := (Config.pPubSubConfig^.PubSubList.pEntries$UDINT + sizeof(t_s_PubSubEntry)*udCount)$^t_s_PubSubEntry;

      if pEntry^.Callback.pThis    &
         pEntry^.Callback.pMethod  then

        pEntry^.Callback.pMethod$PubSub_Callback( pThis       :=  pEntry^.Callback.pThis,
                                                  MsgType     :=  PSRC_Disconnected,
                                                  iMid        :=  -1,
                                                  iGrantedQoS :=  -1,
                                                  pMessage    :=  NIL);

       //If this is the MQTTTopic Class
      elsif pEntry^.Callback.pThis          &
            pEntry^.Callback.pMethod = NIL  then

        pEntry^.Callback.pThis$^MQTTTopic^.PubSubData(MsgType     :=  PSRC_Disconnected,
                                                      iMid        :=  -1,
                                                      iGrantedQoS :=  -1,
                                                      pMessage    :=  NIL);

      end_if;

    end_for;

  end_if;

END_FUNCTION

FUNCTION MQTTClient_Interface::OnPublish
	VAR_INPUT
		mid 	: INT;
	END_VAR
  VAR
  	udCount : UDINT;
    pEntry : ^t_s_PubSubEntry;
    tmpPara : DINT;
  END_VAR

  //If there aren't any Subscribe elements in the Subscribe List | Mem not OK
  if Config.pPubSubConfig^.PubSubList.udNumEntries = 0 then
    //Create Log: Received Publish confirm from MQTTClient without having any elements in the subscription list, ignored.

    tmpPara := to_dint(mid);

    Logging_InterfLog(usLevel     :=  MQTTCLIENTINTERFACE_LOGGING_LEVEL_ERR,
                      dMsgGroup   :=  MQCLIINF_LOG_ERROR_PUBLISH_UNEXPECTED_PUB_CONF_NOTINIT_GRP,
                      dMsgNbr     :=  MQCLIINF_LOG_ERROR_PUBLISH_UNEXPECTED_PUB_CONF_NOTINIT_MSG,
                      pMsg        :=  MQCLIINF_LOG_ERROR_PUBLISH_UNEXPECTED_PUB_CONF_NOTINIT_TEXT,
                      pPara1      :=  #tmpPara,
                      pPara2      :=  NIL,
                      pPara3      :=  NIL,
                      pPara4      :=  NIL);
    return;
  end_if;

  //Step over the entries to find the responsible one
  pEntry := Config.pPubSubConfig^.PubSubList.pEntries;

  for udCount := 0 to Config.pPubSubConfig^.PubSubList.udNumEntries - 1 do

    if pEntry^.iMid = mid &
       pEntry^.EntryType = PSE_Publish then

//      if pEntry^.EntryType <> PSE_Publish then
//        //Create Log: Received a Publish confirmation for a non publish item in the pubsub list, ignored.
//
//        tmpPara := to_dint(mid);
//
//        Logging_InterfLog(usLevel     :=  MQTTCLIENTINTERFACE_LOGGING_LEVEL_WARNING,
//                          dMsgGroup   :=  MQCLIINF_LOG_WARNING_PUBLISH_UNEXP_PUB_CONF_NOT_FOUND_GRP,
//                          dMsgNbr     :=  MQCLIINF_LOG_WARNING_PUBLISH_UNEXP_PUB_CONF_NOT_FOUND_MSG,
//                          pMsg        :=  MQCLIINF_LOG_WARNING_PUBLISH_UNEXP_PUB_CONF_NOT_FOUND_TEXT,
//                          pPara1      :=  #tmpPara,
//                          pPara2      :=  NIL,
//                          pPara3      :=  NIL,
//                          pPara4      :=  NIL);
//
//        //Remove this entry from the PubSub list
//        if Config.pPubSubConfig^.PubSubList.udNumEntries - 1 > udCount then
//
//          SigCLib.MemCpy( dst0  :=  pEntry,
//                          src0  :=  (pEntry$UDINT + sizeof(t_s_PubSubEntry))$^void,
//                          len0  :=  (sizeof(t_s_PubSubEntry) * (Config.pPubSubConfig^.PubSubList.udNumEntries - 1 - udCount)));
//
//        end_if;
//
//        Config.pPubSubConfig^.PubSubList.udNumEntries -= 1;
//
//        return;
//      end_if;

      //If this is a user class
      if pEntry^.Callback.pThis   &
         pEntry^.Callback.pMethod then

        //Call the responsible party.
        pEntry^.Callback.pMethod$PubSub_Callback(pThis        :=  pEntry^.Callback.pThis,
                                                 MsgType      :=  PSRC_Published,
                                                 iMid         :=  mid,
                                                 iGrantedQoS  :=  0,
                                                 pMessage     :=  NIL);
      //If this is the MQTTTopic Class
      elsif pEntry^.Callback.pThis          &
            pEntry^.Callback.pMethod = NIL  then

        pEntry^.Callback.pThis$^MQTTTopic^.PubSubData(MsgType     :=  PSRC_Published,
                                                      iMid        :=  mid,
                                                      iGrantedQoS :=  0,
                                                      pMessage    :=  NIL);

      else
        //Create Log: Received a publish confirmation but could not call back as the Callback parameters weren't OK.

        tmpPara := to_dint(mid);

        Logging_InterfLog(usLevel     :=  MQTTCLIENTINTERFACE_LOGGING_LEVEL_WARNING,
                          dMsgGroup   :=  MQCLIINF_LOG_WARNING_PUBLISH_PUB_CALLBACK_NOTSET_GRP,
                          dMsgNbr     :=  MQCLIINF_LOG_WARNING_PUBLISH_PUB_CALLBACK_NOTSET_MSG,
                          pMsg        :=  MQCLIINF_LOG_WARNING_PUBLISH_PUB_CALLBACK_NOTSET_TEXT,
                          pPara1      :=  #tmpPara,
                          pPara2      :=  NIL,
                          pPara3      :=  NIL,
                          pPara4      :=  NIL);
        return;
      end_if;

      //Remove this entry from the PubSub list
      if Config.pPubSubConfig^.PubSubList.udNumEntries - 1 > udCount then

        SigCLib.MemCpy( dst0  :=  pEntry,
                        src0  :=  (pEntry$UDINT + sizeof(t_s_PubSubEntry))$^void,
                        len0  :=  (sizeof(t_s_PubSubEntry) * (Config.pPubSubConfig^.PubSubList.udNumEntries - 1 - udCount)));

      end_if;
      Config.pPubSubConfig^.PubSubList.udNumEntries -= 1;

      return;

    end_if;

    pEntry$UDINT += sizeof(t_s_PubSubEntry);

  end_for;

  //Create Log: Received publication confirm from MQTTClient and did not find the element in the pubsub list, ignored.

  tmpPara := to_dint(mid);

  Logging_InterfLog(usLevel     :=  MQTTCLIENTINTERFACE_LOGGING_LEVEL_INFO,
                    dMsgGroup   :=  MQCLIINF_LOG_INFO_PUBLISH_PUBLISHED_GRP,
                    dMsgNbr     :=  MQCLIINF_LOG_INFO_PUBLISH_PUBLISHED_MSG,
                    pMsg        :=  MQCLIINF_LOG_INFO_PUBLISH_PUBLISHED_TEXT,
                    pPara1      :=  #tmpPara,
                    pPara2      :=  NIL,
                    pPara3      :=  NIL,
                    pPara4      :=  NIL);

END_FUNCTION

FUNCTION MQTTClient_Interface::OnMessage
	VAR_INPUT
		pMessage 	: ^MQTTClient::t_s_MQTTMessage;
	END_VAR
  VAR
  	udCount : UDINT;
    pSubEntry : ^t_s_PubSubEntry;
    tmpPara : DINT;
  END_VAR

  //Find the Message in the PubSub List and call the responsible party.
  if pMessage then

    //Set the Diagnostic Data
    Diagnostic_Event( Event   :=  DL_RXBytes,
                      udValue :=  pMessage^.payloadlen);

    if Config.pPubSubConfig = NIL then
      //Create Log: Received a published message callback but the pubsublist is not initialised.

      if pMessage <> NIL then
        tmpPara := to_dint(pMessage^.mid);
      else
        tmpPara := 16#FFFF;
      end_if;

      Logging_InterfLog(usLevel     :=  MQTTCLIENTINTERFACE_LOGGING_LEVEL_ERR,
                        dMsgGroup   :=  MQCLIINF_LOG_ERROR_MESSAGE_UNEXPECTED_PUB_CONF_NOTINIT_GRP,
                        dMsgNbr     :=  MQCLIINF_LOG_ERROR_MESSAGE_UNEXPECTED_PUB_CONF_NOTINIT_MSG,
                        pMsg        :=  MQCLIINF_LOG_ERROR_MESSAGE_UNEXPECTED_PUB_CONF_NOTINIT_TEXT,
                        pPara1      :=  #tmpPara,
                        pPara2      :=  NIL,
                        pPara3      :=  NIL,
                        pPara4      :=  NIL);
      return;
    end_if;

    if Config.pPubSubConfig^.PubSubList.udNumEntries = 0 then
      //Create Log: Received a published message callback but the pubsublist is empty.

      if pMessage <> NIL then
        tmpPara := to_dint(pMessage^.mid);
      else
        tmpPara := 16#FFFF;
      end_if;

      Logging_InterfLog(usLevel     :=  MQTTCLIENTINTERFACE_LOGGING_LEVEL_WARNING,
                        dMsgGroup   :=  MQCLIINF_LOG_WARNING_MESSAGE_UNEXP_LIST_EMPTY_GRP,
                        dMsgNbr     :=  MQCLIINF_LOG_WARNING_MESSAGE_UNEXP_LIST_EMPTY_MSG,
                        pMsg        :=  MQCLIINF_LOG_WARNING_MESSAGE_UNEXP_LIST_EMPTY_TEXT,
                        pPara1      :=  #tmpPara,
                        pPara2      :=  NIL,
                        pPara3      :=  NIL,
                        pPara4      :=  NIL);
      return;
    end_if;

    pSubEntry := Config.pPubSubConfig^.PubSubList.pEntries;

    for udCount := 0 to Config.pPubSubConfig^.PubSubList.udNumEntries - 1 do

      if PubSub_TopicCompare(pStr:=pMessage^.topic, pWCString:=#pSubEntry^.aTopic[0])   &
         (pSubEntry^.EntryType = PSE_Subscribe)                                         then

        //If the callback is set call the standard callback
        if pSubEntry^.Callback.pThis    &
           pSubEntry^.Callback.pMethod  then

          pSubEntry^.Callback.pMethod$PubSub_Callback(pThis       :=  pSubEntry^.Callback.pThis,
                                                      MsgType     :=  PSRC_PublishReceived,
                                                      iMid        :=  pMessage^.mid,
                                                      iGrantedQoS :=  0,
                                                      pMessage    :=  pMessage);

        //If this is the MQTTTopic Class, use the class type definition (Allows for Download on the fly)
        elsif pSubEntry^.Callback.pThis          &
              pSubEntry^.Callback.pMethod = NIL  then

          pSubEntry^.Callback.pThis$^MQTTTopic^.PubSubData( MsgType     :=  PSRC_PublishReceived,
                                                            iMid        :=  pMessage^.mid,
                                                            iGrantedQoS :=  0,
                                                            pMessage    :=  pMessage);

        //No Callback is set, this message cannot be delivered
        else

          //Create Log: Received a Published Message Callback but could not call the responsible party as no callback was set

          if pMessage <> NIL then
            tmpPara := to_dint(pMessage^.mid);
          else
            tmpPara := 16#FFFF;
          end_if;

          Logging_InterfLog(usLevel     :=  MQTTCLIENTINTERFACE_LOGGING_LEVEL_WARNING,
                            dMsgGroup   :=  MQCLIINF_LOG_WARNING_MESSAGE_CALLBACK_NOTSET_GRP,
                            dMsgNbr     :=  MQCLIINF_LOG_WARNING_MESSAGE_CALLBACK_NOTSET_MSG,
                            pMsg        :=  MQCLIINF_LOG_WARNING_MESSAGE_CALLBACK_NOTSET_TEXT,
                            pPara1      :=  #tmpPara,
                            pPara2      :=  NIL,
                            pPara3      :=  NIL,
                            pPara4      :=  NIL);

        end_if;

      end_if;

      pSubEntry$UDINT += sizeof(t_s_PubSubEntry);

    end_for;

  end_if;

END_FUNCTION

FUNCTION MQTTClient_Interface::OnSubscribe
	VAR_INPUT
		mid 	: INT;
		qos_count 	: INT;
		granted_qos 	: ^INT;
	END_VAR
  VAR
  	udCount : UDINT;
    pEntry : ^t_s_PubSubEntry;
    tmpPara : DINT;
  END_VAR

  //If there aren't any Subscribe elements in the Subscribe List | Mem not OK
  if  Config.pPubSubConfig = NIL                        |
      Config.pPubSubConfig^.PubSubList.udNumEntries = 0 then
    //Create Log: Received Subscription confirm from MQTTClient without having any elements in the subscription list, ignored.

    tmpPara := to_dint(mid);

    Logging_InterfLog(usLevel     :=  MQTTCLIENTINTERFACE_LOGGING_LEVEL_INFO,
                      dMsgGroup   :=  MQCLIINF_LOG_WARNING_SUBSCRIBE_UNEXP_SUB_CONF_GRP,
                      dMsgNbr     :=  MQCLIINF_LOG_WARNING_SUBSCRIBE_UNEXP_SUB_CONF_MSG,
                      pMsg        :=  MQCLIINF_LOG_WARNING_SUBSCRIBE_UNEXP_SUB_CONF_TEXT,
                      pPara1      :=  #tmpPara,
                      pPara2      :=  #Config.pPubSubConfig^.PubSubList.udNumEntries$DINT,
                      pPara3      :=  NIL,
                      pPara4      :=  NIL);
    return;
  end_if;

  //Step over the entries to find the responsible one
  pEntry := Config.pPubSubConfig^.PubSubList.pEntries;

  for udCount := 0 to Config.pPubSubConfig^.PubSubList.udNumEntries - 1 do

    if pEntry^.iMid = mid &
       pEntry^.EntryType = PSE_Subscribe then

//      if pEntry^.EntryType <> PSE_Subscribe then
//        //Create Log: Received a subscription confirmation for a non subscribe item in the subscription list, ignored.
//
//        tmpPara := to_dint(mid);
//
//        Logging_InterfLog(usLevel     :=  MQTTCLIENTINTERFACE_LOGGING_LEVEL_INFO,
//                          dMsgGroup   :=  MQCLIINF_LOG_WARNING_SUBSCRIBE_SUB_CONF_PUB_ENTRY_GRP,
//                          dMsgNbr     :=  MQCLIINF_LOG_WARNING_SUBSCRIBE_SUB_CONF_PUB_ENTRY_MSG,
//                          pMsg        :=  MQCLIINF_LOG_WARNING_SUBSCRIBE_SUB_CONF_PUB_ENTRY_TEXT,
//                          pPara1      :=  #tmpPara,
//                          pPara2      :=  NIL,
//                          pPara3      :=  NIL,
//                          pPara4      :=  NIL);
//        return;
//      end_if;

      if pEntry^.Callback.pThis &
         pEntry^.Callback.pMethod then

        //Call the responsible party.
        pEntry^.Callback.pMethod$PubSub_Callback(pThis        :=  pEntry^.Callback.pThis,
                                                 MsgType      :=  PSRC_Subscribed,
                                                 iMid         :=  mid,
                                                 iGrantedQoS  :=  granted_qos^,
                                                 pMessage     :=  NIL);

      //If this is the MQTTTopic Class
      elsif pEntry^.Callback.pThis          &
            pEntry^.Callback.pMethod = NIL  then

        pEntry^.Callback.pThis$^MQTTTopic^.PubSubData(MsgType     :=  PSRC_Subscribed,
                                                      iMid        :=  mid,
                                                      iGrantedQoS :=  granted_qos^,
                                                      pMessage    :=  NIL);

      else
        //Create Log: Received a subscription confirmation but could not call back as the Callback parameters weren't OK.

        tmpPara := to_dint(mid);

        Logging_InterfLog(usLevel     :=  MQTTCLIENTINTERFACE_LOGGING_LEVEL_WARNING,
                          dMsgGroup   :=  MQCLIINF_LOG_WARNING_SUBSCRIBE_CALLBACK_NOTSET_GRP,
                          dMsgNbr     :=  MQCLIINF_LOG_WARNING_SUBSCRIBE_CALLBACK_NOTSET_MSG,
                          pMsg        :=  MQCLIINF_LOG_WARNING_SUBSCRIBE_CALLBACK_NOTSET_TEXT,
                          pPara1      :=  #tmpPara,
                          pPara2      :=  NIL,
                          pPara3      :=  NIL,
                          pPara4      :=  NIL);
        return;
      end_if;

      //Stop as we found the element we were interested in.
      return;

    end_if;

    pEntry$UDINT += sizeof(t_s_PubSubEntry);

  end_for;

  //Create Log: Received Subscription confirm from MQTTClient and did not find the element in the subscription list, ignored.

  tmpPara := to_dint(mid);

  Logging_InterfLog(usLevel     :=  MQTTCLIENTINTERFACE_LOGGING_LEVEL_WARNING,
                    dMsgGroup   :=  MQCLIINF_LOG_WARNING_SUBSCRIBE_UNEXP_SUB_CONF_NOT_FOUND_GRP,
                    dMsgNbr     :=  MQCLIINF_LOG_WARNING_SUBSCRIBE_UNEXP_SUB_CONF_NOT_FOUND_MSG,
                    pMsg        :=  MQCLIINF_LOG_WARNING_SUBSCRIBE_UNEXP_SUB_CONF_NOT_FOUND_TEXT,
                    pPara1      :=  #tmpPara,
                    pPara2      :=  NIL,
                    pPara3      :=  NIL,
                    pPara4      :=  NIL);

END_FUNCTION

FUNCTION MQTTClient_Interface::OnUnsubscribe
	VAR_INPUT
		mid 	: INT;
	END_VAR
  VAR
  	udCount : UDINT;
    pEntry : ^t_s_PubSubEntry;
    tmpPara : DINT;
  END_VAR

  //If there aren't any Subscribe elements in the Subscribe List | Mem not OK
  if  Config.pPubSubConfig = NIL                        |
      Config.pPubSubConfig^.PubSubList.udNumEntries = 0 then
    //Create Log: Received UNSUBACK from MQTTClient without having any elements in the subscription list, ignored.

    tmpPara := to_dint(mid);

    Logging_InterfLog(usLevel     :=  MQTTCLIENTINTERFACE_LOGGING_LEVEL_INFO,
                      dMsgGroup   :=  MQCLIINF_LOG_WARNING_UNSUBSCRIBE_UNEXP_LIST_EMPTY_GRP,
                      dMsgNbr     :=  MQCLIINF_LOG_WARNING_UNSUBSCRIBE_UNEXP_LIST_EMPTY_MSG,
                      pMsg        :=  MQCLIINF_LOG_WARNING_UNSUBSCRIBE_UNEXP_LIST_EMPTY_TEXT,
                      pPara1      :=  #tmpPara,
                      pPara2      :=  NIL,
                      pPara3      :=  NIL,
                      pPara4      :=  NIL);
    return;
  end_if;

  //Step over the entries to find the responsible one
  pEntry := Config.pPubSubConfig^.PubSubList.pEntries;

  for udCount := 0 to Config.pPubSubConfig^.PubSubList.udNumEntries - 1 do

    if pEntry^.iUnsubMid = mid &
       pEntry^.EntryType = PSE_Subscribe then

//      if pEntry^.EntryType <> PSE_Subscribe then
//        //Create Log: Received a subscription confirmation for a non subscribe item in the subscription list, ignored.
//
//        tmpPara := to_dint(mid);
//
//        Logging_InterfLog(usLevel     :=  MQTTCLIENTINTERFACE_LOGGING_LEVEL_WARNING,
//                          dMsgGroup   :=  MQCLIINF_LOG_WARNING_UNSUBSCRIBE_WRONG_ENTRY_GRP,
//                          dMsgNbr     :=  MQCLIINF_LOG_WARNING_UNSUBSCRIBE_WRONG_ENTRY_MSG,
//                          pMsg        :=  MQCLIINF_LOG_WARNING_UNSUBSCRIBE_WRONG_ENTRY_TEXT,
//                          pPara1      :=  #tmpPara,
//                          pPara2      :=  NIL,
//                          pPara3      :=  NIL,
//                          pPara4      :=  NIL);
//        return;
//      end_if;

      if pEntry^.Callback.pThis &
         pEntry^.Callback.pMethod then

        //Call the responsible party.
        pEntry^.Callback.pMethod$PubSub_Callback(pThis        :=  pEntry^.Callback.pThis,
                                                 MsgType      :=  PSRC_Unsubscribed,
                                                 iMid         :=  mid,
                                                 iGrantedQoS  :=  -1,
                                                 pMessage     :=  NIL);

       //If this is the MQTTTopic Class
        elsif pEntry^.Callback.pThis          &
              pEntry^.Callback.pMethod = NIL  then

          pEntry^.Callback.pThis$^MQTTTopic^.PubSubData(MsgType     :=  PSRC_Unsubscribed,
                                                        iMid        :=  mid,
                                                        iGrantedQoS :=  -1,
                                                        pMessage    :=  NIL);

      else
        //Create Log: Received an unsubscription confirmation but could not call back as the Callback parameters weren't OK.

        tmpPara := to_dint(mid);

        Logging_InterfLog(usLevel     :=  MQTTCLIENTINTERFACE_LOGGING_LEVEL_WARNING,
                          dMsgGroup   :=  MQCLIINF_LOG_WARNING_UNSUBSCRIBE_CALLBACK_NOTSET_GRP,
                          dMsgNbr     :=  MQCLIINF_LOG_WARNING_UNSUBSCRIBE_CALLBACK_NOTSET_MSG,
                          pMsg        :=  MQCLIINF_LOG_WARNING_UNSUBSCRIBE_CALLBACK_NOTSET_TEXT,
                          pPara1      :=  #tmpPara,
                          pPara2      :=  NIL,
                          pPara3      :=  NIL,
                          pPara4      :=  NIL);
      end_if;

      //Remove this entry from the PubSub list
      if Config.pPubSubConfig^.PubSubList.udNumEntries - 1 > udCount then

        SigCLib.MemCpy( dst0  :=  pEntry,
                          src0  :=  (pEntry$UDINT + sizeof(t_s_PubSubEntry))$^void,
                          len0  :=  (sizeof(t_s_PubSubEntry) * (Config.pPubSubConfig^.PubSubList.udNumEntries - 1 - udCount)));

      end_if;

      Config.pPubSubConfig^.PubSubList.udNumEntries -= 1;

      return;

    end_if;

    pEntry$UDINT += sizeof(t_s_PubSubEntry);

  end_for;

  //Create Log: Received Subscription confirm from MQTTClient and did not find the element in the subscription list, ignored.

  tmpPara := to_dint(mid);

  Logging_InterfLog(usLevel     :=  MQTTCLIENTINTERFACE_LOGGING_LEVEL_INFO,
                    dMsgGroup   :=  MQCLIINF_LOG_INFO_UNSUBSCRIBE_UNSUBSCRIBED_GRP,
                    dMsgNbr     :=  MQCLIINF_LOG_INFO_UNSUBSCRIBE_UNSUBSCRIBED_MSG,
                    pMsg        :=  MQCLIINF_LOG_INFO_UNSUBSCRIBE_UNSUBSCRIBED_TEXT,
                    pPara1      :=  #tmpPara,
                    pPara2      :=  NIL,
                    pPara3      :=  NIL,
                    pPara4      :=  NIL);

END_FUNCTION

FUNCTION MQTTClient_Interface::OnLog
	VAR_INPUT
		level 	: INT;
		pStr 	: ^CHAR;
	END_VAR
  VAR
  	dLogLevel : DINT;
  END_VAR

  //If the string pointer is not OK, Log and stop
  if pStr = NIL then

    dLogLevel := to_dint(level);

    //Log Failure
    Logging_InterfLog(usLevel     :=  MQTTCLIENTINTERFACE_LOGGING_LEVEL_ERR,
                      dMsgGroup   :=  MQCLIINF_LOG_ERROR_LOGGING_NO_TEXT_GRP,
                      dMsgNbr     :=  MQCLIINF_LOG_ERROR_LOGGING_NO_TEXT_MSG,
                      pMsg        :=  MQCLIINF_LOG_ERROR_LOGGING_NO_TEXT_TEXT,
                      pPara1      :=  #dLogLevel,
                      pPara2      :=  NIL,
                      pPara3      :=  NIL,
                      pPara4      :=  NIL);
    return;

  end_if;

  //Diagnostic info
  Diagnostic_Event( Event   :=  DL_Log,
                    udValue :=  0);

  //====================================================
  //Decide the Application Log Level based on MQTT Level
  //====================================================
  case level of
    //-------------------
    //Info -> Info
    //-------------------
    MQTT_LOG_INFO:
      dLogLevel := MQTTCLIENTINTERFACE_LOGGING_LEVEL_INFO;
    //-------------------
    //Notice -> Info
    //-------------------
    MQTT_LOG_NOTICE:
      dLogLevel := MQTTCLIENTINTERFACE_LOGGING_LEVEL_INFO;
    //-------------------
    //Warning -> Warning
    //-------------------
    MQTT_LOG_WARNING:
      dLogLevel := MQTTCLIENTINTERFACE_LOGGING_LEVEL_WARNING;
    //-------------------
    //Error -> Error
    //-------------------
    MQTT_LOG_ERR:
      dLogLevel := MQTTCLIENTINTERFACE_LOGGING_LEVEL_ERR;
    //-------------------
    //Debug -> Debug
    //-------------------
    MQTT_LOG_DEBUG:
      dLogLevel := MQTTCLIENTINTERFACE_LOGGING_LEVEL_DEBUG;

  else

    dLogLevel := to_dint(level);

    //Log Failure
    Logging_InterfLog(usLevel     :=  MQTTCLIENTINTERFACE_LOGGING_LEVEL_ERR,
                      dMsgGroup   :=  MQCLIINF_LOG_ERROR_LOGGING_UNKNOWN_LEVEL_GRP,
                      dMsgNbr     :=  MQCLIINF_LOG_ERROR_LOGGING_UNKNOWN_LEVEL_MSG,
                      pMsg        :=  MQCLIINF_LOG_ERROR_LOGGING_UNKNOWN_LEVEL_TEXT,
                      pPara1      :=  #dLogLevel,
                      pPara2      :=  NIL,
                      pPara3      :=  NIL,
                      pPara4      :=  NIL);
    return;

  end_case;

  //Log Message from MQTTClient
  Logging_InterfLog(usLevel     :=  to_usint(dLogLevel),
                    dMsgGroup   :=  MQTTCLIENTINTERFACE_LOG_MQTTCLIENT_MSGGRP,
                    dMsgNbr     :=  MQTTCLIENTINTERFACE_LOG_MQTTCLIENT_MSGNBR,
                    pMsg        :=  pStr,
                    pPara1      :=  NIL,
                    pPara2      :=  NIL,
                    pPara3      :=  NIL,
                    pPara4      :=  NIL);

END_FUNCTION

FUNCTION MQTTClient_Interface::OnLog_WithDetail
	VAR_INPUT
		usLevel 	  : USINT;
		dMsgGroup 	: DINT;
		dMsgNbr 	  : DINT;
		pMsg 	      : ^CHAR;
		pPara1 	    : ^DINT;
		pPara2 	    : ^DINT;
		pPara3 	    : ^DINT;
		pPara4 	    : ^DINT;
	END_VAR
  VAR
  	dLogLevel : DINT;
  END_VAR

  //===================================
  //Set the Last Log Details
  //===================================
  case usLevel of

    //-----------------
    //Error
    //-----------------
    MQTT_LOG_ERR:

      DiagnosticData.LogEvents.Level_Error.dLastClientGroup   := dMsgGroup;
      DiagnosticData.LogEvents.Level_Error.dLastClientMessage := dMsgNbr;

      DiagnosticData.LogEvents.Level_Error.dLastGlobalGroup   := dMsgGroup;
      DiagnosticData.LogEvents.Level_Error.dLastGlobalMessage := dMsgNbr;

    //-----------------
    //Info
    //-----------------
    MQTT_LOG_INFO:

      DiagnosticData.LogEvents.Level_Info.dLastClientGroup   := dMsgGroup;
      DiagnosticData.LogEvents.Level_Info.dLastClientMessage := dMsgNbr;

      DiagnosticData.LogEvents.Level_Info.dLastGlobalGroup   := dMsgGroup;
      DiagnosticData.LogEvents.Level_Info.dLastGlobalMessage := dMsgNbr;

    //-----------------
    //Debug
    //-----------------
    MQTT_LOG_DEBUG:

      DiagnosticData.LogEvents.Level_Debug.dLastClientGroup   := dMsgGroup;
      DiagnosticData.LogEvents.Level_Debug.dLastClientMessage := dMsgNbr;

      DiagnosticData.LogEvents.Level_Debug.dLastGlobalGroup   := dMsgGroup;
      DiagnosticData.LogEvents.Level_Debug.dLastGlobalMessage := dMsgNbr;

    //-----------------
    //Warning
    //-----------------
    MQTT_LOG_WARNING:

      DiagnosticData.LogEvents.Level_Warning.dLastClientGroup   := dMsgGroup;
      DiagnosticData.LogEvents.Level_Warning.dLastClientMessage := dMsgNbr;

      DiagnosticData.LogEvents.Level_Warning.dLastGlobalGroup   := dMsgGroup;
      DiagnosticData.LogEvents.Level_Warning.dLastGlobalMessage := dMsgNbr;

  end_case;

  //If the string pointer is not OK, Log and stop
  if pMsg = NIL then

    dLogLevel := to_dint(uslevel);

    //Log Failure
    Logging_InternLog(usLevel     :=  MQTTCLIENTINTERFACE_LOGGING_LEVEL_ERR,
                      dMsgGroup   :=  MQCLIINF_LOG_ERROR_LOGGING_NO_TEXT_GRP,
                      dMsgNbr     :=  MQCLIINF_LOG_ERROR_LOGGING_NO_TEXT_MSG,
                      pMsg        :=  MQCLIINF_LOG_ERROR_LOGGING_NO_TEXT_TEXT,
                      pPara1      :=  #dLogLevel,
                      pPara2      :=  NIL,
                      pPara3      :=  NIL,
                      pPara4      :=  NIL);
    return;

  end_if;

  //Diagnostic info
  Diagnostic_Event( Event   :=  DL_Log,
                    udValue :=  0);

  //Log Message from MQTTClient
  Logging_InternLog(usLevel     :=  usLevel,
                    dMsgGroup   :=  dMsgGroup,
                    dMsgNbr     :=  dMsgNbr,
                    pMsg        :=  pMsg,
                    pPara1      :=  pPara1,
                    pPara2      :=  pPara2,
                    pPara3      :=  pPara3,
                    pPara4      :=  pPara4, 1);

END_FUNCTION

//================================================================================================================================================================
//-------------------------------------------------------------------END OF CALLBACK METHODS----------------------------------------------------------------------
//================================================================================================================================================================

//================================================================================================================================================================
//-------------------------------------------------------------------------COUNTER METHODS------------------------------------------------------------------------
//================================================================================================================================================================
FUNCTION MQTTClient_Interface::Counters_IncSubMID
	VAR_OUTPUT
		iMid 	: INT;
	END_VAR

  Config.iNextSubMID += 1;

  if Config.iNextSubMID >= MQTTCLIENTINTERFACE_SUB_MID_ROLLOVER then
    Config.iNextSubMID := MQTTCLIENTINTERFACE_SUB_MID_INITVAL;
  end_if;

  iMid := Config.iNextSubMID;

END_FUNCTION

FUNCTION MQTTClient_Interface::Counters_GetSubMID
	VAR_OUTPUT
		iMID 	: INT;
	END_VAR

  iMID := Config.iNextSubMID;

END_FUNCTION

FUNCTION MQTTClient_Interface::Counters_IncPubMID
	VAR_OUTPUT
		iMid 	: INT;
	END_VAR

  Config.iNextPubMID += 1;

  if Config.iNextPubMID >= MQTTCLIENTINTERFACE_PUB_MID_ROLLOVER then
    Config.iNextPubMID := MQTTCLIENTINTERFACE_PUB_MID_INITVAL;
  end_if;

  iMid := Config.iNextPubMID;

END_FUNCTION

FUNCTION MQTTClient_Interface::Counters_GetPubMID
	VAR_OUTPUT
		iMID 	: INT;
	END_VAR

  iMID := Config.iNextPubMID;

END_FUNCTION

FUNCTION MQTTClient_Interface::Counters_IncApplID
	VAR_OUTPUT
		udApplID 	: UDINT;
	END_VAR

  udApplID := 0;

  if Config.pPubSubConfig = NIL then
    return;
  end_if;

  Config.pPubSubConfig^.udNextAppliID += 1;

  if Config.pPubSubConfig^.udNextAppliID > MQTTCLIENTINTERFACE_APPLID_ROLLOVER then
    Config.pPubSubConfig^.udNextAppliID := MQTTCLIENTINTERFACE_APPLID_INITVAL;
  end_if;

  udApplID := Config.pPubSubConfig^.udNextAppliID;

END_FUNCTION

FUNCTION MQTTClient_Interface::Counters_GetApplID
	VAR_OUTPUT
		udApplID 	: UDINT;
	END_VAR

  udApplID := 0;

  if Config.pPubSubConfig then
    udApplID := Config.pPubSubConfig^.udNextAppliID;
  end_if;

END_FUNCTION

//================================================================================================================================================================
//---------------------------------------------------------------------END OF COUNTER METHODS---------------------------------------------------------------------
//================================================================================================================================================================

FUNCTION GLOBAL MQTTClient_Interface::MQTT_ReadLogConfig
	VAR_OUTPUT
		bUpdated 	: BOOL;
	END_VAR

  bUpdated := FALSE;

  if Config.IsConn.LogConfig then
    cLogConfig := cLogConfig.Read();
    bUpdated := TRUE;
  end_if;

END_FUNCTION

FUNCTION VIRTUAL GLOBAL MQTTClient_Interface::CleanSession::Read
	VAR_OUTPUT
		output (EAX) 	: DINT;
	END_VAR

	CleanSession := MQTTClient.CleanSession.Read();
	output := CleanSession;

END_FUNCTION

FUNCTION VIRTUAL GLOBAL MQTTClient_Interface::CleanSession::Write
	VAR_INPUT
		input (EAX) 	: DINT;
	END_VAR
	VAR_OUTPUT
		result (EAX) 	: DINT;
	END_VAR

	CleanSession := input;
	result := (MQTTClient.CleanSession.Write(CleanSession))$DINT;

END_FUNCTION

FUNCTION VIRTUAL GLOBAL MQTTClient_Interface::SessionPresent::Read
	VAR_OUTPUT
		output (EAX) 	: DINT;
	END_VAR

	SessionPresent := MQTTClient.SessionPresent.Read();
	output := SessionPresent;

END_FUNCTION

FUNCTION MQTTClient_Interface::PubSub_TopicCompare
	VAR_INPUT
		pStr 	: ^UINT;
		pWCString 	: ^UINT;
	END_VAR
	VAR_OUTPUT
		bEqual 	: BOOL;
	END_VAR
  VAR
  	pTopic, pWCTopic : ^UINT;
  END_VAR

  //Assume that the strings are not equal
  bEqual := FALSE;

  //If the input is OK, continue the comparison
  if pStr      &
     pWCString then

    pTopic    := pStr;
    pWCTopic  := pWCString;

    //Special case: The Wildcard string starts with the Multi-Layer Wildcard -> Immediately matches.
    if pWCTopic^ = MQTTCLIENTINTERFACE_TOPIC_WC_MULTI then
      bEqual := TRUE;
      return;
    end_if;

    while (pWCTopic^ = pTopic^)                             |
          (pWCTopic^ = MQTTCLIENTINTERFACE_TOPIC_WC_MULTI)  |
          (pWCTopic^ = MQTTCLIENTINTERFACE_TOPIC_WC_SINGLE) do

      //Found a Multi-layer Wildcard - The topics are equal (We don't confirm that nothing follows the #).
      if pWCTopic^ = MQTTCLIENTINTERFACE_TOPIC_WC_MULTI then

        bEqual := TRUE;
        return;

      //Found a single layer wildcard - Skip this Topic Layer
      elsif pWCTopic^ = MQTTCLIENTINTERFACE_TOPIC_WC_SINGLE then

        while pTopic^ <> MQTTCLIENTINTERFACE_TOPIC_SEPARATOR  &
              pTopic^ <> 0$UINT                               do
          pTopic$UDINT += sizeof(UINT);
        end_while;

        pWCTopic$UDINT += sizeof(UINT);

        //Special Case: WC-String ended on a + -> (text/+ = text/topic)
        if pWCTopic^ = 0$UINT then

          if pTopic^ = MQTTCLIENTINTERFACE_TOPIC_SEPARATOR then
            pTopic$UDINT += sizeof(UINT);
          end_if;

          if pTopic^ = pWCTopic^ then
            bEqual := TRUE;
          end_if;

          return;

        end_if;

      //If we have reached the end of the string, stop
      elsif pWCTopic^ = 0$UINT then

        bEqual := TRUE;
        return;

      end_if;

      //Advance the String pointers
      pTopic$UDINT    += sizeof(UINT);
      pWCTopic$UDINT  += sizeof(UINT);

      //If either String ends but the other continues, the topics aren't equal
      if (pTopic^ = 0$UINT &
          pWCTopic^ <> 0$UINT)  |
         (pWCTopic^ = 0$UINT &
          pTopic^ <> 0$UINT)    then
        return;
      end_if;

      //Jump over Separators
      if pTopic^ = MQTTCLIENTINTERFACE_TOPIC_SEPARATOR then
        pTopic$UDINT    += sizeof(UINT);
      end_if;

      if pWCTopic^ = MQTTCLIENTINTERFACE_TOPIC_SEPARATOR then
        pWCTopic$UDINT    += sizeof(UINT);
      end_if;

    end_while;

  end_if;

END_FUNCTION

FUNCTION MQTTClient_Interface::PubSub_Reset
  VAR
  	udCount : UDINT;
    pEntry : ^t_s_PubSubEntry;
  END_VAR

  //Step through the Subscribed entites and send the Unsubscribed callback
  if Config.pPubSubConfig &
     Config.pPubSubConfig^.PubSubList.udNumEntries > 0 then

    for udCount := 0 to Config.pPubSubConfig^.PubSubList.udNumEntries - 1 do

      pEntry := (Config.pPubSubConfig^.PubSubList.pEntries$UDINT + sizeof(t_s_PubSubEntry)*udCount)$^t_s_PubSubEntry;

      if pEntry^.EntryType = PSE_Subscribe then

        //If the callback method is set call the method
        if pEntry^.Callback.pThis    &
           pEntry^.Callback.pMethod  then

          pEntry^.Callback.pMethod$PubSub_Callback( pThis       :=  pEntry^.Callback.pThis,
                                                    MsgType     :=  PSRC_Unsubscribed,
                                                    iMid        :=  -1,
                                                    iGrantedQoS :=  -1,
                                                    pMessage    :=  NIL);
        //If this is the MQTTTopic Class
        elsif pEntry^.Callback.pThis          &
              pEntry^.Callback.pMethod = NIL  then

          pEntry^.Callback.pThis$^MQTTTopic^.PubSubData(MsgType     :=  PSRC_Unsubscribed,
                                                        iMid        :=  -1,
                                                        iGrantedQoS :=  -1,
                                                        pMessage    :=  NIL);

        end_if;

      end_if;
    end_for;

    Config.pPubSubConfig^.PubSubList.udNumEntries := 0;
    sigclib_memset( dst :=  Config.pPubSubConfig^.PubSubList.pEntries,
                    c   :=  0x00,
                    len :=  Config.pPubSubConfig^.PubSubList.udMaxEntries * sizeof(t_s_PubSubEntry));

  end_if;

END_FUNCTION

FUNCTION MQTTClient_Interface::PubSub_CheckSubscription
	VAR_INPUT
		pTopic 	: ^UINT;
		pThis 	: ^void;
		pCallback 	: ^void;
	END_VAR
	VAR_OUTPUT
		udAppliID 	: UDINT;
	END_VAR
  VAR
  	udCount : UDINT;
    pEntry : ^t_s_PubSubEntry;
  END_VAR

  udAppliID := 0;

  if Config.pPubSubConfig &
     Config.pPubSubConfig^.PubSubList.udNumEntries > 0 then

    for udCount := 0 to Config.pPubSubConfig^.PubSubList.udNumEntries - 1 do

      pEntry := (Config.pPubSubConfig^.PubSubList.pEntries$UDINT + udCount*sizeof(t_s_PubSubEntry))$^t_s_PubSubEntry;

      if pEntry^.Callback.pMethod = pCallback           &
         pEntry^.Callback.pThis   = pThis               &
         sigclib_strcmp16(src1  :=  #pEntry^.aTopic[0],
                          src2  :=  pTopic) = 0         then

        udAppliID := pEntry^.udAppliID;
        return;

      end_if;

    end_for;

  end_if;

  return;

END_FUNCTION

FUNCTION MQTTClient_Interface::Diagnostic_Calculate
  VAR
    udCount : UDINT;
  END_VAR

  //If the Calculation Interval has passed, update the diagnostic information
  if ops.tAbsolute - DiagnosticData.udLastCalcTimestamp >= MQTTCLIENTINTERFACE_DIAGNOSTIC_TX_RATE_CALCINTERVAL then

    //=======================================================
    //Transfer Rate Calc
    //=======================================================

      //Input current Transfer Rates
      DiagnosticData.TransferRateCalc.aTxEntries[DiagnosticData.TransferRateCalc.udIndex] := DiagnosticData.ComDiagnosis.udTotalBytesTx - DiagnosticData.TransferRateCalc.udLastTotalBytesTx;
      DiagnosticData.TransferRateCalc.aRxEntries[DiagnosticData.TransferRateCalc.udIndex] := DiagnosticData.ComDiagnosis.udTotalBytesRx - DiagnosticData.TransferRateCalc.udLastTotalBytesRx;

      DiagnosticData.TransferRateCalc.udLastTotalBytesTx := DiagnosticData.ComDiagnosis.udTotalBytesTx;
      DiagnosticData.TransferRateCalc.udLastTotalBytesRx := DiagnosticData.ComDiagnosis.udTotalBytesRx;

      //Adjust index
      DiagnosticData.TransferRateCalc.udIndex   += 1;
      if DiagnosticData.TransferRateCalc.udIndex = MQTTCLIENTINTERFACE_DIAGNOSTIC_TX_RATE_CALC_AVG then
        DiagnosticData.TransferRateCalc.udIndex := 0;
      end_if;

      //Calculate current average
      DiagnosticData.ComDiagnosis.udTxRate := DiagnosticData.ComDiagnosis.udRxRate := 0;

      for udCount := 0 to MQTTCLIENTINTERFACE_DIAGNOSTIC_TX_RATE_CALC_AVG - 1 do
        DiagnosticData.ComDiagnosis.udTxRate += DiagnosticData.TransferRateCalc.aTxEntries[udCount];
        DiagnosticData.ComDiagnosis.udRxRate += DiagnosticData.TransferRateCalc.aRxEntries[udCount];
      end_for;

      //Set the rate values
      Diagnostic_Event( Event   :=  DL_TXRate,
                        udValue :=  to_udint(to_real(DiagnosticData.ComDiagnosis.udTxRate)/to_real(MQTTCLIENTINTERFACE_DIAGNOSTIC_TX_RATE_CALC_AVG)));
      Diagnostic_Event( Event   :=  DL_RXRate,
                        udValue :=  to_udint(to_real(DiagnosticData.ComDiagnosis.udRxRate)/to_real(MQTTCLIENTINTERFACE_DIAGNOSTIC_TX_RATE_CALC_AVG)));

    //=======================================================
    //PubSub List Counts
    //=======================================================

      //PubsUbList Entries
      if Config.pPubSubConfig then
        Diagnostic_Event( Event   :=  DL_PubSubEntries,
                          udValue :=  Config.pPubSubConfig^.PubSubList.udNumEntries);
      else
        Diagnostic_Event( Event   :=  DL_PubSubEntries,
                          udValue :=  0);
      end_if;

    //=======================================================
    //DataMap List Counts
    //=======================================================

      //DataMap Entries
      if Config.pDataMapConfig then

        Diagnostic_Event( Event   :=  DL_DataMapEntries,
                          udValue :=  Config.pDataMapConfig^.udPublishElements + Config.pDataMapConfig^.udSubscribeElements);

      else

        Diagnostic_Event( Event   :=  DL_DataMapEntries,
                          udValue :=  0);

      end_if;

    DiagnosticData.udLastCalcTimestamp := ops.tAbsolute;

  end_if;

END_FUNCTION

FUNCTION VIRTUAL GLOBAL MQTTClient_Interface::ComDiagnosis::NewInst
	VAR_INPUT
		pPara 	: ^CmdStruct;
		pResult 	: ^Results;
	END_VAR
	VAR_OUTPUT
		ret_code 	: IprStates;
	END_VAR

  if  pPara = NIL |
      pResult = NIL then
    ret_code := ERROR;
    return;
  end_if;

	CASE pPara^.uiCmd OF
		MQTTCLIENTINTERFACE_DIAGNOSTIC_NEWINST_COMDIAG_ID : Diagnostic_GetData( pPara   :=  pPara,
                                                                            pResult :=  pResult);
	END_CASE;

	ret_code := READY;

END_FUNCTION

FUNCTION MQTTClient_Interface::Diagnostic_GetData
	VAR_INPUT
		pPara 	: ^CmdStruct;
		pResult 	: ^results;
	END_VAR

  //==============================================================
  //Based on the diagnostic command, perform the required task
  //==============================================================
  case pPara^.aPara[1] of
    //-------------------------------------------------------------
    //Reset All Values
    //-------------------------------------------------------------
    MQTTCLIENTINTERFACE_DIAGNOSTIC_NEWINST_COMDIAG_RESET:

      Diagnostic_Event( Event   :=  DL_Reset,
                        udValue :=  0);

    //-------------------------------------------------------------
    //Number of Connection Attempts
    //-------------------------------------------------------------
    MQTTCLIENTINTERFACE_DIAGNOSTIC_NEWINST_GET_CONNECTCOUNT:

      pResult^.aData[0]$UDINT := DiagnosticData.ComDiagnosis.udConnect;

    //-------------------------------------------------------------
    //Number of Failed Connections
    //-------------------------------------------------------------
    MQTTCLIENTINTERFACE_DIAGNOSTIC_NEWINST_GET_CONNECTFAILCNT:

      pResult^.aData[0]$UDINT := DiagnosticData.ComDiagnosis.udConnectFail;

    //-------------------------------------------------------------
    //Number of Connection Retries
    //-------------------------------------------------------------
    MQTTCLIENTINTERFACE_DIAGNOSTIC_NEWINST_GET_RETRYCOUNT:

      pResult^.aData[0]$UDINT := DiagnosticData.ComDiagnosis.udConnectRetry;

    //-------------------------------------------------------------
    //Number of Connection Watchdog Timeouts
    //-------------------------------------------------------------
    MQTTCLIENTINTERFACE_DIAGNOSTIC_NEWINST_GET_WATCHDOGCOUNT:

      pResult^.aData[0]$UDINT := DiagnosticData.ComDiagnosis.udWDTimeout;

    //-------------------------------------------------------------
    //Not Used
    //-------------------------------------------------------------
    MQTTCLIENTINTERFACE_DIAGNOSTIC_NEWINST_GET_ACTERRORCODE:

      pResult^.aData[0]$UDINT := 0;

    //-------------------------------------------------------------
    //Last Non Successful Return Value from MQTTClient
    //-------------------------------------------------------------
    MQTTCLIENTINTERFACE_DIAGNOSTIC_NEWINST_GET_LASTERRORCODE:

      pResult^.aData[0]$UDINT := DiagnosticData.ComDiagnosis.udLastRet;

    //-------------------------------------------------------------
    //Number of non successful returns from MQTTClient
    //-------------------------------------------------------------
    MQTTCLIENTINTERFACE_DIAGNOSTIC_NEWINST_GET_ERRORCNT:

      pResult^.aData[0]$UDINT := DiagnosticData.ComDiagnosis.udFailRet;

    //-------------------------------------------------------------
    //Number of Subscribe Requests
    //-------------------------------------------------------------
    MQTTCLIENTINTERFACE_DIAGNOSTIC_NEWINST_GET_READCNT:

      pResult^.aData[0]$UDINT := DiagnosticData.ComDiagnosis.udSubReqs;

    //-------------------------------------------------------------
    //Number of Subscribe Failures
    //-------------------------------------------------------------
    MQTTCLIENTINTERFACE_DIAGNOSTIC_NEWINST_GET_READERRORCNT:

      pResult^.aData[0]$UDINT := DiagnosticData.ComDiagnosis.udSubFail;

    //-------------------------------------------------------------
    //Number of Publish Requests
    //-------------------------------------------------------------
    MQTTCLIENTINTERFACE_DIAGNOSTIC_NEWINST_GET_WRITECNT:

      pResult^.aData[0]$UDINT := DiagnosticData.ComDiagnosis.udPubReq;

    //-------------------------------------------------------------
    //Number of Publish Failures
    //-------------------------------------------------------------
    MQTTCLIENTINTERFACE_DIAGNOSTIC_NEWINST_GET_WRITEERRORCNT:

      pResult^.aData[0]$UDINT := DiagnosticData.ComDiagnosis.udPubFail;

    //-------------------------------------------------------------
    //Number of Unsubscribe Requests
    //-------------------------------------------------------------
    MQTTCLIENTINTERFACE_DIAGNOSTIC_NEWINST_GET_UNSUBSCRIBES:

      pResult^.aData[0]$UDINT := DiagnosticData.ComDiagnosis.udUnsubReq;

    //-------------------------------------------------------------
    //Number of Unsubscribe Failures
    //-------------------------------------------------------------
    MQTTCLIENTINTERFACE_DIAGNOSTIC_NEWINST_GET_UNSUBFAILS:

      pResult^.aData[0]$UDINT := DiagnosticData.ComDiagnosis.udUnsubFail;

    //-------------------------------------------------------------
    //Number of PubSub List Entries
    //-------------------------------------------------------------
    MQTTCLIENTINTERFACE_DIAGNOSTIC_NEWINST_GET_PUBSUBENTRIES:

      pResult^.aData[0]$UDINT := DiagnosticData.ComDiagnosis.udPubSubEntries;

    //-------------------------------------------------------------
    //Number of Logs Made
    //-------------------------------------------------------------
    MQTTCLIENTINTERFACE_DIAGNOSTIC_NEWINST_GET_LOGCOUNT:

      pResult^.aData[0]$UDINT := DiagnosticData.ComDiagnosis.udLogs;

    //-------------------------------------------------------------
    //Number of PINGREQ Sent
    //-------------------------------------------------------------
    MQTTCLIENTINTERFACE_DIAGNOSTIC_NEWINST_GET_PINGREQSENT:

      pResult^.aData[0]$UDINT := DiagnosticData.ComDiagnosis.udPingReq;

    //-------------------------------------------------------------
    //Number of PINGRESP Received
    //-------------------------------------------------------------
    MQTTCLIENTINTERFACE_DIAGNOSTIC_NEWINST_GET_PINGRESPREC:

      pResult^.aData[0]$UDINT := DiagnosticData.ComDiagnosis.udPingResp;

    //-------------------------------------------------------------
    //Number of QOS0 Publish Messages
    //-------------------------------------------------------------
    MQTTCLIENTINTERFACE_DIAGNOSTIC_NEWINST_GET_QOS0_PUB:

      pResult^.aData[0]$UDINT := DiagnosticData.ComDiagnosis.udPubQOS0;

    //-------------------------------------------------------------
    //Number of QOS1 Publish Messages
    //-------------------------------------------------------------
    MQTTCLIENTINTERFACE_DIAGNOSTIC_NEWINST_GET_QOS1_PUB:

      pResult^.aData[0]$UDINT := DiagnosticData.ComDiagnosis.udPubQOS1;

    //-------------------------------------------------------------
    //Number of QOS2 Publish Messages
    //-------------------------------------------------------------
    MQTTCLIENTINTERFACE_DIAGNOSTIC_NEWINST_GET_QOS2_PUB:

      pResult^.aData[0]$UDINT := DiagnosticData.ComDiagnosis.udPubQOS2;

    //-------------------------------------------------------------
    //Number of QOS0 Subscribe Messages
    //-------------------------------------------------------------
    MQTTCLIENTINTERFACE_DIAGNOSTIC_NEWINST_GET_QOS0_SUB:

      pResult^.aData[0]$UDINT := DiagnosticData.ComDiagnosis.udSubQOS0;

    //-------------------------------------------------------------
    //Number of QOS1 Subscribe Messages
    //-------------------------------------------------------------
    MQTTCLIENTINTERFACE_DIAGNOSTIC_NEWINST_GET_QOS1_SUB:

      pResult^.aData[0]$UDINT := DiagnosticData.ComDiagnosis.udSubQOS1;

    //-------------------------------------------------------------
    //Number of QOS2 Subscribe Messages
    //-------------------------------------------------------------
    MQTTCLIENTINTERFACE_DIAGNOSTIC_NEWINST_GET_QOS2_SUB:

      pResult^.aData[0]$UDINT := DiagnosticData.ComDiagnosis.udSubQOS2;

    //-------------------------------------------------------------
    //Number of Datamap Entries
    //-------------------------------------------------------------
    MQTTCLIENTINTERFACE_DIAGNOSTIC_NEWINST_GET_DM_ELEMENTS:
